C09133=1217.822,182.147,-55.204,-177.681,6.059,148.397
C09134=1217.818,182.396,-55.226,-177.678,6.061,148.396
C09135=1217.814,182.645,-55.250,-177.676,6.062,148.396
C09136=1217.809,182.894,-55.272,-177.674,6.064,148.396
C09137=1217.804,183.143,-55.295,-177.670,6.066,148.395
C09138=1217.799,183.392,-55.318,-177.668,6.067,148.395
C09139=1217.795,183.641,-55.340,-177.666,6.068,148.394
C09140=1217.790,183.890,-55.364,-177.663,6.070,148.394
C09141=1217.785,184.139,-55.387,-177.660,6.072,148.394
C09142=1217.781,184.387,-55.409,-177.658,6.074,148.393
C09143=1217.776,184.636,-55.433,-177.655,6.075,148.393
C09144=1217.772,184.886,-55.455,-177.652,6.076,148.392
C09145=1217.767,185.155,-55.480,-177.650,6.078,148.392
C09146=1217.762,185.425,-55.506,-177.647,6.080,148.392
C09147=1217.757,185.694,-55.530,-177.644,6.082,148.391
C09148=1217.752,185.964,-55.555,-177.641,6.083,148.391
C09149=1217.747,186.213,-55.578,-177.639,6.085,148.390
C09150=1217.742,186.461,-55.600,-177.636,6.087,148.390
C09151=1217.738,186.710,-55.623,-177.634,6.088,148.390
C09152=1217.733,186.960,-55.647,-177.631,6.090,148.389
C09153=1217.728,187.209,-55.670,-177.628,6.091,148.389
C09154=1217.724,187.457,-55.693,-177.626,6.093,148.388
C09155=1217.720,187.706,-55.716,-177.623,6.095,148.388
C09156=1217.715,187.955,-55.740,-177.621,6.096,148.388
C09157=1217.710,188.203,-55.762,-177.618,6.098,148.387
C09158=1217.706,188.452,-55.785,-177.615,6.100,148.387
C09159=1217.701,188.701,-55.809,-177.613,6.102,148.387
C09160=1217.696,188.950,-55.832,-177.611,6.103,148.386
C09161=1217.692,189.199,-55.855,-177.608,6.104,148.386
C09162=1217.688,189.448,-55.878,-177.605,6.106,148.385
C09163=1217.683,189.697,-55.902,-177.602,6.108,148.385
C09164=1217.678,189.946,-55.925,-177.600,6.110,148.385
C09165=1217.673,190.195,-55.948,-177.598,6.111,148.384
C09166=1217.668,190.444,-55.971,-177.595,6.112,148.384
C09167=1217.664,190.692,-55.994,-177.592,6.114,148.384
C09168=1217.660,190.941,-56.017,-177.590,6.116,148.383
C09169=1217.655,191.190,-56.041,-177.587,6.118,148.383
C09170=1217.650,191.439,-56.064,-177.585,6.119,148.382
C09171=1217.645,191.688,-56.088,-177.582,6.120,148.382
C09172=1217.641,191.938,-56.111,-177.579,6.122,148.382
C09173=1217.637,192.186,-56.134,-177.576,6.124,148.381
C09174=1217.632,192.435,-56.158,-177.574,6.126,148.381
C09175=1217.628,192.684,-56.181,-177.572,6.127,148.380
C09176=1217.622,192.932,-56.204,-177.569,6.129,148.380
C09177=1217.618,193.181,-56.227,-177.566,6.131,148.380
C09178=1217.613,193.430,-56.251,-177.564,6.132,148.379
C09179=1217.608,193.679,-56.274,-177.561,6.134,148.379
C09180=1217.604,193.928,-56.298,-177.559,6.135,148.379
C09181=1217.599,194.177,-56.322,-177.556,6.137,148.378
C09182=1217.595,194.425,-56.344,-177.553,6.139,148.378
C09183=1217.591,194.674,-56.368,-177.551,6.140,148.377
C09184=1217.586,194.923,-56.391,-177.548,6.142,148.377
C09185=1217.581,195.172,-56.415,-177.545,6.144,148.377
C09186=1217.577,195.421,-56.439,-177.543,6.145,148.376
C09187=1217.572,195.670,-56.462,-177.541,6.147,148.376
C09188=1217.567,195.919,-56.485,-177.538,6.149,148.376
C09189=1217.563,196.167,-56.509,-177.535,6.151,148.375
C09190=1217.558,196.416,-56.533,-177.533,6.152,148.375
C09191=1217.554,196.665,-56.556,-177.530,6.154,148.375
C09192=1217.549,196.914,-56.580,-177.528,6.155,148.374
C09193=1217.544,197.163,-56.603,-177.525,6.157,148.374
C09194=1217.540,197.412,-56.627,-177.523,6.159,148.374
C09195=1217.535,197.660,-56.651,-177.520,6.161,148.373
C09196=1217.531,197.909,-56.674,-177.517,6.163,148.373
C09197=1217.526,198.158,-56.698,-177.514,6.164,148.372
C09198=1217.522,198.407,-56.722,-177.512,6.165,148.372
C09199=1217.517,198.656,-56.745,-177.510,6.167,148.372
C09200=1217.512,198.905,-56.768,-177.507,6.169,148.371
C09201=1217.508,199.153,-56.792,-177.504,6.171,148.371
C09202=1217.504,199.403,-56.816,-177.502,6.173,148.371
C09203=1217.499,199.651,-56.840,-177.499,6.174,148.370
C09204=1217.494,199.901,-56.864,-177.497,6.175,148.370
C09205=1217.489,200.149,-56.888,-177.494,6.177,148.370
C09206=1217.485,200.398,-56.912,-177.492,6.179,148.369
C09207=1217.480,200.647,-56.936,-177.489,6.181,148.369
C09208=1217.476,200.896,-56.959,-177.486,6.183,148.368
C09209=1217.471,201.144,-56.983,-177.484,6.185,148.368
C09210=1217.467,201.393,-57.007,-177.481,6.186,148.368
C09211=1217.462,201.641,-57.031,-177.478,6.188,148.367
C09212=1217.457,201.890,-57.054,-177.476,6.189,148.367
C09213=1217.452,202.139,-57.079,-177.474,6.191,148.367
C09214=1217.448,202.389,-57.102,-177.471,6.193,148.366
C09215=1217.444,202.637,-57.126,-177.468,6.195,148.366
C09216=1217.439,202.886,-57.150,-177.466,6.197,148.366
C09217=1217.435,203.135,-57.174,-177.463,6.198,148.365
C09218=1217.430,203.383,-57.198,-177.460,6.200,148.365
C09219=1217.425,203.633,-57.222,-177.458,6.202,148.365
C09220=1217.421,203.881,-57.246,-177.456,6.203,148.364
C09221=1217.416,204.130,-57.269,-177.453,6.205,148.364
C09222=1217.412,204.379,-57.294,-177.450,6.207,148.364
C09223=1217.408,204.627,-57.318,-177.448,6.209,148.363
C09224=1217.402,204.877,-57.342,-177.445,6.211,148.363
C09225=1217.398,205.125,-57.366,-177.442,6.212,148.363
C09226=1217.393,205.374,-57.390,-177.440,6.214,148.362
C09227=1217.389,205.623,-57.413,-177.437,6.216,148.362
C09228=1217.384,205.872,-57.438,-177.435,6.217,148.362
C09229=1217.380,206.121,-57.462,-177.432,6.219,148.361
C09230=1217.375,206.370,-57.486,-177.429,6.220,148.361
C09231=1217.371,206.618,-57.510,-177.427,6.222,148.360
C09232=1217.366,206.867,-57.535,-177.424,6.224,148.360
C09233=1217.362,207.116,-57.559,-177.421,6.226,148.360
C09234=1217.357,207.365,-57.582,-177.419,6.228,148.359
C09235=1217.352,207.614,-57.607,-177.417,6.230,148.359
C09236=1217.348,207.862,-57.631,-177.414,6.232,148.359
C09237=1217.343,208.110,-57.655,-177.411,6.234,148.359
C09238=1217.339,208.359,-57.680,-177.409,6.235,148.358
C09239=1217.334,208.609,-57.704,-177.407,6.236,148.358
C09240=1217.330,208.857,-57.728,-177.404,6.238,148.358
C09241=1217.324,209.106,-57.752,-177.401,6.240,148.357
C09242=1217.320,209.354,-57.776,-177.399,6.242,148.357
C09243=1217.316,209.603,-57.801,-177.396,6.244,148.357
C09244=1217.311,209.852,-57.825,-177.393,6.246,148.356
C09245=1217.307,210.101,-57.850,-177.391,6.248,148.356
C09246=1217.302,210.349,-57.874,-177.388,6.249,148.355
C09247=1217.297,210.599,-57.898,-177.386,6.251,148.355
C09248=1217.293,210.848,-57.922,-177.383,6.253,148.355
C09249=1217.288,211.118,-57.949,-177.380,6.255,148.354
C09250=1217.283,211.388,-57.975,-177.377,6.256,148.354
C09251=1217.278,211.659,-58.002,-177.375,6.258,148.354
C09252=1217.273,211.929,-58.028,-177.372,6.260,148.353
C09253=1217.268,212.178,-58.053,-177.369,6.262,148.353
C09254=1217.264,212.426,-58.077,-177.367,6.264,148.353
C09255=1217.259,212.676,-58.102,-177.364,6.266,148.352
C09256=1217.255,212.924,-58.126,-177.361,6.268,148.352
C09257=1217.250,213.173,-58.150,-177.359,6.269,148.352
C09258=1217.246,213.422,-58.175,-177.356,6.271,148.351
C09259=1217.241,213.671,-58.200,-177.353,6.273,148.351
C09260=1217.237,213.919,-58.224,-177.351,6.275,148.351
C09261=1217.232,214.168,-58.249,-177.348,6.277,148.350
C09262=1217.228,214.416,-58.273,-177.346,6.279,148.350
C09263=1217.223,214.665,-58.298,-177.343,6.281,148.350
C09264=1217.219,214.914,-58.323,-177.341,6.283,148.349
C09265=1217.214,215.163,-58.347,-177.338,6.285,148.349
C09266=1217.209,215.411,-58.371,-177.335,6.286,148.349
C09267=1217.205,215.661,-58.396,-177.333,6.288,148.348
C09268=1217.201,215.909,-58.420,-177.330,6.290,148.348
C09269=1217.195,216.158,-58.445,-177.328,6.292,148.348
C09270=1217.192,216.406,-58.470,-177.325,6.294,148.347
C09271=1217.187,216.655,-58.495,-177.322,6.296,148.347
C09272=1217.182,216.904,-58.519,-177.320,6.297,148.347
C09273=1217.178,217.153,-58.544,-177.318,6.298,148.346
C09274=1217.173,217.402,-58.569,-177.315,6.300,148.346
C09275=1217.169,217.650,-58.594,-177.312,6.302,148.346
C09276=1217.164,217.899,-58.618,-177.310,6.304,148.345
C09277=1217.160,218.147,-58.643,-177.307,6.306,148.345
C09278=1217.155,218.397,-58.668,-177.305,6.308,148.345
C09279=1217.150,218.645,-58.693,-177.302,6.310,148.345
C09280=1217.147,218.894,-58.717,-177.300,6.312,148.344
C09281=1217.141,219.143,-58.742,-177.297,6.314,148.344
C09282=1217.136,219.391,-58.767,-177.294,6.315,148.344
C09283=1217.133,219.640,-58.792,-177.292,6.317,148.343
C09284=1217.128,219.889,-58.817,-177.289,6.319,148.343
C09285=1217.123,220.138,-58.842,-177.286,6.321,148.343
C09286=1217.119,220.386,-58.866,-177.284,6.323,148.342
C09287=1217.115,220.635,-58.891,-177.281,6.325,148.342
C09288=1217.109,220.884,-58.916,-177.279,6.327,148.342
C09289=1217.105,221.132,-58.941,-177.276,6.329,148.342
C09290=1217.101,221.381,-58.966,-177.274,6.331,148.341
C09291=1217.096,221.629,-58.991,-177.271,6.332,148.341
C09292=1217.092,221.878,-59.016,-177.269,6.334,148.341
C09293=1217.087,222.127,-59.040,-177.266,6.336,148.340
C09294=1217.083,222.376,-59.066,-177.263,6.338,148.340
C09295=1217.078,222.625,-59.091,-177.261,6.340,148.340
C09296=1217.074,222.873,-59.116,-177.258,6.342,148.339
C09297=1217.069,223.122,-59.141,-177.255,6.344,148.339
C09298=1217.065,223.371,-59.166,-177.253,6.346,148.339
C09299=1217.060,223.619,-59.191,-177.251,6.348,148.339
C09300=1217.056,223.868,-59.216,-177.248,6.349,148.338
C09301=1217.051,224.117,-59.241,-177.245,6.351,148.338
C09302=1217.047,224.365,-59.267,-177.243,6.353,148.338
C09303=1217.042,224.614,-59.291,-177.240,6.355,148.337
C09304=1217.038,224.863,-59.317,-177.237,6.357,148.337
C09305=1217.033,225.111,-59.341,-177.235,6.359,148.337
C09306=1217.029,225.360,-59.367,-177.233,6.361,148.337
C09307=1217.024,225.609,-59.392,-177.230,6.363,148.336
C09308=1217.020,225.858,-59.417,-177.227,6.365,148.336
C09309=1217.014,226.106,-59.442,-177.225,6.366,148.336
C09310=1217.010,226.355,-59.468,-177.222,6.368,148.335
C09311=1217.005,226.603,-59.493,-177.219,6.370,148.335
C09312=1217.002,226.852,-59.518,-177.217,6.372,148.335
C09313=1216.997,227.101,-59.543,-177.215,6.374,148.334
C09314=1216.993,227.349,-59.569,-177.212,6.376,148.334
C09315=1216.988,227.599,-59.594,-177.209,6.378,148.334
C09316=1216.983,227.847,-59.619,-177.207,6.380,148.333
C09317=1216.979,228.096,-59.645,-177.204,6.382,148.333
C09318=1216.974,228.344,-59.670,-177.202,6.383,148.333
C09319=1216.970,228.593,-59.695,-177.199,6.386,148.333
C09320=1216.965,228.842,-59.721,-177.197,6.387,148.332
C09321=1216.961,229.090,-59.745,-177.194,6.389,148.332
C09322=1216.957,229.339,-59.771,-177.192,6.391,148.332
C09323=1216.952,229.587,-59.796,-177.189,6.393,148.331
C09324=1216.948,229.836,-59.822,-177.186,6.395,148.331
C09325=1216.943,230.086,-59.847,-177.184,6.397,148.331
C09326=1216.938,230.334,-59.872,-177.182,6.399,148.331
C09327=1216.934,230.582,-59.898,-177.179,6.401,148.330
C09328=1216.929,230.831,-59.924,-177.176,6.403,148.330
C09329=1216.925,231.079,-59.949,-177.174,6.405,148.330
C09330=1216.921,231.329,-59.974,-177.171,6.406,148.329
C09331=1216.916,231.577,-60.000,-177.169,6.409,148.329
C09332=1216.911,231.826,-60.026,-177.166,6.410,148.329
C09333=1216.907,232.075,-60.051,-177.164,6.412,148.329
C09334=1216.902,232.323,-60.077,-177.161,6.414,148.328
C09335=1216.898,232.571,-60.102,-177.158,6.417,148.328
C09336=1216.894,232.820,-60.128,-177.156,6.419,148.328
C09337=1216.889,233.069,-60.153,-177.153,6.421,148.328
C09338=1216.885,233.318,-60.179,-177.150,6.423,148.327
C09339=1216.880,233.567,-60.205,-177.148,6.425,148.327
C09340=1216.875,233.815,-60.230,-177.145,6.426,148.327
C09341=1216.871,234.064,-60.256,-177.143,6.429,148.327
C09342=1216.866,234.313,-60.282,-177.140,6.430,148.326
C09343=1216.862,234.561,-60.307,-177.138,6.432,148.326
C09344=1216.857,234.809,-60.333,-177.135,6.434,148.326
C09345=1216.853,235.058,-60.359,-177.133,6.436,148.326
C09346=1216.848,235.306,-60.384,-177.130,6.438,148.325
C09347=1216.844,235.555,-60.410,-177.128,6.440,148.325
C09348=1216.840,235.804,-60.436,-177.125,6.442,148.325
C09349=1216.835,236.053,-60.462,-177.122,6.444,148.324
C09350=1216.830,236.301,-60.487,-177.120,6.446,148.324
C09351=1216.826,236.550,-60.513,-177.118,6.448,148.324
C09352=1216.822,236.799,-60.539,-177.115,6.450,148.324
C09353=1216.817,237.069,-60.567,-177.112,6.452,148.323
C09354=1216.812,237.341,-60.595,-177.109,6.454,148.323
C09355=1216.807,237.613,-60.623,-177.107,6.456,148.323
C09356=1216.802,237.884,-60.652,-177.103,6.459,148.322
C09357=1216.797,238.133,-60.678,-177.101,6.461,148.322
C09358=1216.793,238.382,-60.704,-177.099,6.463,148.322
C09359=1216.788,238.630,-60.729,-177.096,6.465,148.322
C09360=1216.784,238.879,-60.755,-177.093,6.467,148.321
C09361=1216.780,239.127,-60.781,-177.091,6.469,148.321
C09362=1216.775,239.376,-60.808,-177.089,6.471,148.321
C09363=1216.771,239.625,-60.833,-177.086,6.473,148.321
C09364=1216.766,239.873,-60.859,-177.083,6.474,148.320
C09365=1216.761,240.122,-60.885,-177.081,6.477,148.320
C09366=1216.757,240.371,-60.911,-177.079,6.478,148.320
C09367=1216.753,240.619,-60.937,-177.076,6.481,148.320
C09368=1216.749,240.868,-60.963,-177.073,6.483,148.319
C09369=1216.743,241.116,-60.989,-177.071,6.485,148.319
C09370=1216.739,241.365,-61.015,-177.068,6.487,148.319
C09371=1216.735,241.613,-61.041,-177.066,6.489,148.319
C09372=1216.730,241.862,-61.068,-177.063,6.491,148.318
C09373=1216.726,242.111,-61.093,-177.061,6.493,148.318
C09374=1216.721,242.359,-61.120,-177.058,6.495,148.318
C09375=1216.716,242.608,-61.146,-177.056,6.497,148.317
C09376=1216.712,242.856,-61.172,-177.053,6.499,148.317
C09377=1216.708,243.105,-61.198,-177.051,6.501,148.317
C09378=1216.703,243.354,-61.224,-177.048,6.503,148.317
C09379=1216.699,243.603,-61.250,-177.045,6.505,148.316
C09380=1216.695,243.851,-61.277,-177.043,6.507,148.316
C09381=1216.690,244.099,-61.303,-177.040,6.509,148.316
C09382=1216.686,244.347,-61.329,-177.038,6.511,148.316
C09383=1216.681,244.596,-61.355,-177.035,6.513,148.316
C09384=1216.676,244.845,-61.381,-177.033,6.515,148.315
C09385=1216.673,245.093,-61.408,-177.030,6.517,148.315
C09386=1216.668,245.343,-61.434,-177.028,6.519,148.315
C09387=1216.664,245.591,-61.460,-177.025,6.521,148.315
C09388=1216.659,245.840,-61.487,-177.022,6.524,148.314
C09389=1216.655,246.088,-61.513,-177.020,6.526,148.314
C09390=1216.650,246.336,-61.539,-177.017,6.528,148.314
C09391=1216.645,246.585,-61.566,-177.015,6.530,148.314
C09392=1216.641,246.833,-61.592,-177.012,6.532,148.313
C09393=1216.636,247.082,-61.619,-177.010,6.534,148.313
C09394=1216.632,247.331,-61.644,-177.007,6.536,148.313
C09395=1216.628,247.579,-61.671,-177.005,6.538,148.313
C09396=1216.623,247.828,-61.697,-177.002,6.541,148.313
C09397=1216.619,248.077,-61.724,-177.000,6.542,148.312
C09398=1216.615,248.325,-61.751,-176.997,6.544,148.312
C09399=1216.610,248.574,-61.777,-176.995,6.547,148.312
C09400=1216.606,248.822,-61.803,-176.992,6.548,148.312
C09401=1216.601,249.071,-61.830,-176.990,6.550,148.311
C09402=1216.597,249.319,-61.856,-176.987,6.552,148.311
C09403=1216.592,249.568,-61.883,-176.985,6.554,148.311
C09404=1216.588,249.817,-61.909,-176.982,6.557,148.311
C09405=1216.583,250.065,-61.936,-176.980,6.559,148.310
C09406=1216.579,250.314,-61.963,-176.977,6.561,148.310
C09407=1216.575,250.562,-61.989,-176.974,6.563,148.310
C09408=1216.570,250.811,-62.016,-176.972,6.565,148.310
C09409=1216.565,251.058,-62.042,-176.970,6.567,148.309
C09410=1216.561,251.307,-62.069,-176.966,6.570,148.309
C09411=1216.557,251.556,-62.095,-176.964,6.572,148.309
C09412=1216.552,251.805,-62.122,-176.962,6.574,148.309
C09413=1216.548,252.053,-62.149,-176.959,6.576,148.308
C09414=1216.544,252.302,-62.176,-176.957,6.578,148.308
C09415=1216.539,252.551,-62.202,-176.954,6.580,148.308
C09416=1216.534,252.799,-62.229,-176.952,6.582,148.308
C09417=1216.530,253.047,-62.256,-176.949,6.585,148.308
C09418=1216.526,253.296,-62.283,-176.946,6.586,148.307
C09419=1216.521,253.544,-62.310,-176.944,6.589,148.307
C09420=1216.517,253.793,-62.336,-176.942,6.591,148.307
C09421=1216.512,254.042,-62.363,-176.939,6.592,148.307
C09422=1216.507,254.290,-62.390,-176.937,6.595,148.307
C09423=1216.504,254.538,-62.416,-176.934,6.597,148.306
C09424=1216.499,254.787,-62.443,-176.931,6.599,148.306
C09425=1216.494,255.035,-62.470,-176.929,6.601,148.306
C09426=1216.490,255.284,-62.497,-176.926,6.603,148.306
C09427=1216.486,255.532,-62.524,-176.924,6.605,148.306
C09428=1216.481,255.781,-62.550,-176.922,6.607,148.305
C09429=1216.476,256.030,-62.577,-176.919,6.610,148.305
C09430=1216.472,256.278,-62.604,-176.916,6.612,148.305
C09431=1216.468,256.527,-62.631,-176.914,6.614,148.305
C09432=1216.463,256.776,-62.658,-176.911,6.616,148.305
C09433=1216.459,257.024,-62.685,-176.909,6.618,148.304
C09434=1216.455,257.272,-62.712,-176.906,6.621,148.304
C09435=1216.450,257.521,-62.739,-176.904,6.623,148.304
C09436=1216.446,257.769,-62.766,-176.901,6.625,148.304
C09437=1216.441,258.018,-62.793,-176.899,6.627,148.303
C09438=1216.436,258.266,-62.820,-176.896,6.629,148.303
C09439=1216.432,258.514,-62.846,-176.893,6.632,148.303
C09440=1216.429,258.763,-62.875,-176.891,6.634,148.303
C09441=1216.424,259.011,-62.902,-176.888,6.636,148.303
C09442=1216.419,259.260,-62.929,-176.886,6.638,148.302
C09443=1216.415,259.508,-62.956,-176.884,6.640,148.302
C09444=1216.410,259.757,-62.983,-176.881,6.643,148.302
C09445=1216.406,260.005,-63.009,-176.878,6.645,148.302
C09446=1216.401,260.254,-63.036,-176.876,6.647,148.302
C09447=1216.397,260.503,-63.064,-176.873,6.649,148.301
C09448=1216.393,260.751,-63.091,-176.871,6.651,148.301
C09449=1216.388,260.999,-63.119,-176.868,6.654,148.301
C09450=1216.384,261.248,-63.146,-176.866,6.656,148.301
C09451=1216.379,261.496,-63.173,-176.863,6.658,148.301
C09452=1216.375,261.745,-63.200,-176.861,6.660,148.300
C09453=1216.370,261.994,-63.227,-176.859,6.662,148.300
C09454=1216.367,262.241,-63.254,-176.856,6.664,148.300
C09455=1216.362,262.490,-63.282,-176.853,6.667,148.300
C09456=1216.357,262.738,-63.309,-176.851,6.669,148.300
C09457=1216.353,263.012,-63.339,-176.848,6.671,148.299
C09458=1216.348,263.284,-63.369,-176.845,6.673,148.299
C09459=1216.343,263.557,-63.399,-176.842,6.676,148.299
C09460=1216.338,263.829,-63.429,-176.840,6.678,148.299
C09461=1216.334,264.077,-63.456,-176.838,6.680,148.299
C09462=1216.330,264.327,-63.483,-176.834,6.683,148.298
C09463=1216.325,264.575,-63.511,-176.832,6.685,148.298
C09464=1216.321,264.823,-63.538,-176.830,6.687,148.298
C09465=1216.316,265.072,-63.565,-176.828,6.689,148.298
C09466=1216.312,265.320,-63.594,-176.824,6.692,148.298
C09467=1216.308,265.569,-63.621,-176.822,6.694,148.298
C09468=1216.303,265.817,-63.648,-176.820,6.696,148.297
C09469=1216.299,266.065,-63.675,-176.817,6.698,148.297
C09470=1216.294,266.315,-63.703,-176.814,6.701,148.297
C09471=1216.289,266.562,-63.731,-176.812,6.703,148.297
C09472=1216.285,266.811,-63.758,-176.810,6.705,148.297
C09473=1216.280,267.059,-63.785,-176.807,6.707,148.297
C09474=1216.276,267.308,-63.814,-176.804,6.710,148.296
C09475=1216.272,267.556,-63.841,-176.802,6.712,148.296
C09476=1216.267,267.804,-63.868,-176.800,6.714,148.296
C09477=1216.263,268.054,-63.896,-176.797,6.716,148.296
C09478=1216.259,268.301,-63.924,-176.794,6.719,148.296
C09479=1216.254,268.550,-63.951,-176.792,6.721,148.296
C09480=1216.251,268.798,-63.979,-176.790,6.723,148.295
C09481=1216.245,269.047,-64.006,-176.787,6.725,148.295
C09482=1216.241,269.295,-64.034,-176.784,6.728,148.295
C09483=1216.236,269.543,-64.062,-176.782,6.730,148.295
C09484=1216.232,269.792,-64.089,-176.779,6.732,148.295
C09485=1216.228,270.040,-64.117,-176.777,6.735,148.294
C09486=1216.224,270.289,-64.145,-176.774,6.737,148.294
C09487=1216.219,270.537,-64.173,-176.772,6.739,148.294
C09488=1216.215,270.785,-64.201,-176.769,6.741,148.294
C09489=1216.210,271.035,-64.228,-176.767,6.744,148.294
C09490=1216.206,271.282,-64.256,-176.764,6.746,148.293
C09491=1216.201,271.531,-64.283,-176.762,6.748,148.293
C09492=1216.197,271.780,-64.312,-176.760,6.750,148.293
C09493=1216.193,272.028,-64.340,-176.757,6.753,148.293
C09494=1216.188,272.276,-64.367,-176.755,6.755,148.293
C09495=1216.184,272.525,-64.395,-176.752,6.757,148.293
C09496=1216.179,272.773,-64.423,-176.749,6.760,148.293
C09497=1216.175,273.022,-64.451,-176.747,6.762,148.292
C09498=1216.171,273.270,-64.478,-176.745,6.764,148.292
C09499=1216.166,273.518,-64.506,-176.742,6.766,148.292
C09500=1216.162,273.767,-64.535,-176.739,6.769,148.292
C09501=1216.158,274.015,-64.563,-176.737,6.771,148.292
C09502=1216.153,274.264,-64.590,-176.735,6.773,148.292
C09503=1216.149,274.512,-64.618,-176.732,6.776,148.292
C09504=1216.145,274.761,-64.647,-176.729,6.778,148.291
C09505=1216.140,275.008,-64.674,-176.727,6.780,148.291
C09506=1216.136,275.256,-64.702,-176.724,6.783,148.291
C09507=1216.131,275.505,-64.731,-176.722,6.785,148.291
C09508=1216.127,275.754,-64.758,-176.720,6.787,148.291
C09509=1216.123,276.002,-64.786,-176.717,6.789,148.291
C09510=1216.118,276.250,-64.814,-176.714,6.792,148.290
C09511=1216.114,276.499,-64.843,-176.712,6.794,148.290
C09512=1216.109,276.747,-64.871,-176.710,6.796,148.290
C09513=1216.105,276.996,-64.899,-176.707,6.799,148.290
C09514=1216.101,277.244,-64.927,-176.704,6.801,148.290
C09515=1216.097,277.493,-64.956,-176.702,6.803,148.290
C09516=1216.092,277.740,-64.983,-176.699,6.806,148.289
C09517=1216.088,277.989,-65.011,-176.697,6.808,148.289
C09518=1216.083,278.237,-65.040,-176.695,6.811,148.289
C09519=1216.080,278.486,-65.068,-176.692,6.813,148.289
C09520=1216.074,278.734,-65.096,-176.690,6.815,148.289
C09521=1216.071,278.983,-65.125,-176.687,6.818,148.289
C09522=1216.066,279.231,-65.153,-176.684,6.820,148.289
C09523=1216.062,279.479,-65.181,-176.682,6.823,148.289
C09524=1216.058,279.727,-65.209,-176.680,6.824,148.288
C09525=1216.053,279.976,-65.238,-176.677,6.827,148.288
C09526=1216.049,280.224,-65.265,-176.675,6.830,148.288
C09527=1216.044,280.473,-65.294,-176.672,6.832,148.288
C09528=1216.040,280.721,-65.322,-176.669,6.835,148.288
C09529=1216.035,280.970,-65.351,-176.667,6.837,148.288
C09530=1216.031,281.218,-65.378,-176.665,6.839,148.288
C09531=1216.027,281.466,-65.407,-176.662,6.842,148.288
C09532=1216.023,281.715,-65.435,-176.660,6.844,148.287
C09533=1216.018,281.963,-65.464,-176.657,6.846,148.287
C09534=1216.014,282.211,-65.492,-176.655,6.849,148.287
C09535=1216.009,282.459,-65.521,-176.653,6.851,148.287
C09536=1216.005,282.708,-65.550,-176.650,6.853,148.287
C09537=1216.000,282.956,-65.577,-176.647,6.856,148.287
C09538=1215.996,283.204,-65.607,-176.645,6.858,148.287
C09539=1215.992,283.453,-65.635,-176.643,6.860,148.286
C09540=1215.987,283.701,-65.663,-176.640,6.863,148.286
C09541=1215.984,283.950,-65.691,-176.638,6.865,148.286
C09542=1215.978,284.198,-65.720,-176.635,6.868,148.286
C09543=1215.974,284.446,-65.749,-176.632,6.870,148.286
C09544=1215.971,284.695,-65.777,-176.630,6.872,148.286
C09545=1215.965,284.943,-65.806,-176.628,6.875,148.286
C09546=1215.961,285.191,-65.835,-176.625,6.877,148.286
C09547=1215.957,285.439,-65.863,-176.623,6.879,148.286
C09548=1215.952,285.688,-65.892,-176.620,6.883,148.286
C09549=1215.948,285.936,-65.921,-176.618,6.884,148.285
C09550=1215.944,286.184,-65.949,-176.616,6.887,148.285
C09551=1215.939,286.433,-65.978,-176.613,6.890,148.285
C09552=1215.935,286.681,-66.007,-176.611,6.892,148.285
C09553=1215.931,286.929,-66.035,-176.608,6.895,148.285
C09554=1215.926,287.178,-66.064,-176.605,6.897,148.285
C09555=1215.922,287.426,-66.093,-176.603,6.899,148.285
C09556=1215.918,287.674,-66.121,-176.600,6.902,148.284
C09557=1215.914,287.922,-66.150,-176.598,6.904,148.284
C09558=1215.909,288.171,-66.179,-176.596,6.906,148.284
C09559=1215.905,288.419,-66.208,-176.593,6.909,148.284
C09560=1215.901,288.667,-66.236,-176.591,6.911,148.284
C09561=1215.896,288.942,-66.268,-176.588,6.914,148.284
C09562=1215.891,289.216,-66.300,-176.585,6.917,148.284
C09563=1215.887,289.490,-66.332,-176.583,6.919,148.284
C09564=1215.882,289.764,-66.364,-176.580,6.922,148.284
C09565=1215.878,290.013,-66.393,-176.577,6.925,148.284
C09566=1215.872,290.261,-66.421,-176.575,6.927,148.283
C09567=1215.868,290.509,-66.451,-176.573,6.929,148.283
C09568=1215.864,290.758,-66.480,-176.570,6.932,148.283
C09569=1215.860,291.006,-66.509,-176.568,6.934,148.283
C09570=1215.855,291.254,-66.537,-176.565,6.937,148.283
C09571=1215.851,291.502,-66.566,-176.563,6.939,148.283
C09572=1215.847,291.751,-66.596,-176.560,6.942,148.283
C09573=1215.842,291.999,-66.625,-176.558,6.945,148.283
C09574=1215.838,292.247,-66.654,-176.556,6.947,148.283
C09575=1215.834,292.495,-66.682,-176.553,6.950,148.283
C09576=1215.830,292.744,-66.711,-176.550,6.952,148.283
C09577=1215.826,292.992,-66.741,-176.548,6.954,148.282
C09578=1215.821,293.240,-66.770,-176.546,6.957,148.282
C09579=1215.816,293.489,-66.798,-176.543,6.959,148.282
C09580=1215.812,293.737,-66.828,-176.541,6.962,148.282
C09581=1215.808,293.985,-66.857,-176.538,6.964,148.282
C09582=1215.803,294.234,-66.886,-176.536,6.966,148.282
C09583=1215.799,294.482,-66.915,-176.533,6.969,148.282
C09584=1215.795,294.729,-66.944,-176.531,6.972,148.282
C09585=1215.791,294.978,-66.974,-176.529,6.975,148.282
C09586=1215.787,295.227,-67.002,-176.526,6.977,148.282
C09587=1215.782,295.475,-67.032,-176.524,6.979,148.282
C09588=1215.778,295.722,-67.061,-176.521,6.982,148.282
C09589=1215.773,295.971,-67.090,-176.519,6.984,148.281
C09590=1215.769,296.219,-67.120,-176.516,6.987,148.281
C09591=1215.765,296.467,-67.149,-176.514,6.989,148.281
C09592=1215.761,296.716,-67.178,-176.512,6.992,148.281
C09593=1215.756,296.964,-67.207,-176.509,6.994,148.281
C09594=1215.752,297.212,-67.236,-176.507,6.996,148.281
C09595=1215.747,297.460,-67.266,-176.504,6.999,148.281
C09596=1215.743,297.709,-67.295,-176.502,7.001,148.281
C09597=1215.739,297.957,-67.325,-176.499,7.005,148.281
C09598=1215.735,298.205,-67.354,-176.497,7.007,148.281
C09599=1215.731,298.453,-67.384,-176.495,7.010,148.281
C09600=1215.726,298.702,-67.413,-176.492,7.012,148.281
C09601=1215.722,298.950,-67.443,-176.490,7.014,148.281
C09602=1215.718,299.197,-67.472,-176.488,7.017,148.281
C09603=1215.713,299.446,-67.501,-176.485,7.019,148.280
C09604=1215.709,299.694,-67.531,-176.482,7.022,148.280
C09605=1215.704,299.943,-67.561,-176.480,7.024,148.280
C09606=1215.700,300.191,-67.590,-176.478,7.027,148.280
C09607=1215.696,300.439,-67.620,-176.476,7.030,148.280
C09608=1215.692,300.687,-67.649,-176.473,7.033,148.280
C09609=1215.688,300.936,-67.678,-176.471,7.035,148.280
C09610=1215.683,301.184,-67.708,-176.469,7.037,148.280
C09611=1215.679,301.432,-67.737,-176.466,7.040,148.280
C09612=1215.675,301.680,-67.767,-176.464,7.042,148.280
C09613=1215.670,301.928,-67.796,-176.461,7.045,148.280
C09614=1215.665,302.177,-67.826,-176.459,7.048,148.280
C09615=1215.661,302.425,-67.855,-176.456,7.051,148.280
C09616=1215.657,302.673,-67.885,-176.454,7.053,148.280
C09617=1215.653,302.921,-67.914,-176.452,7.056,148.280
C09618=1215.649,303.169,-67.945,-176.449,7.058,148.280
C09619=1215.644,303.418,-67.975,-176.447,7.060,148.280
C09620=1215.640,303.666,-68.004,-176.444,7.063,148.280
C09621=1215.636,303.914,-68.033,-176.442,7.065,148.280
C09622=1215.631,304.162,-68.063,-176.439,7.068,148.280
C09623=1215.628,304.410,-68.093,-176.437,7.070,148.280
C09624=1215.623,304.659,-68.123,-176.435,7.073,148.280
C09625=1215.618,304.907,-68.153,-176.432,7.076,148.279
C09626=1215.614,305.155,-68.182,-176.430,7.079,148.279
C09627=1215.610,305.403,-68.212,-176.428,7.081,148.279
C09628=1215.605,305.651,-68.242,-176.425,7.084,148.279
C09629=1215.601,305.900,-68.272,-176.423,7.086,148.279
C09630=1215.597,306.148,-68.301,-176.420,7.089,148.279
C09631=1215.592,306.396,-68.332,-176.418,7.091,148.279
C09632=1215.588,306.644,-68.361,-176.416,7.094,148.279
C09633=1215.584,306.892,-68.391,-176.413,7.097,148.279
C09634=1215.580,307.140,-68.421,-176.412,7.099,148.279
C09635=1215.575,307.389,-68.451,-176.409,7.102,148.279
C09636=1215.571,307.637,-68.481,-176.407,7.104,148.279
C09637=1215.567,307.885,-68.511,-176.404,7.107,148.279
C09638=1215.562,308.133,-68.541,-176.402,7.110,148.279
C09639=1215.558,308.381,-68.571,-176.399,7.113,148.279
C09640=1215.554,308.629,-68.601,-176.397,7.115,148.279
C09641=1215.549,308.878,-68.630,-176.395,7.118,148.279
C09642=1215.545,309.125,-68.661,-176.393,7.120,148.279
C09643=1215.541,309.375,-68.691,-176.390,7.123,148.279
C09644=1215.537,309.622,-68.721,-176.388,7.125,148.279
C09645=1215.533,309.870,-68.751,-176.385,7.128,148.279
C09646=1215.528,310.118,-68.781,-176.383,7.131,148.279
C09647=1215.524,310.367,-68.811,-176.381,7.133,148.279
C09648=1215.520,310.615,-68.842,-176.378,7.136,148.279
C09649=1215.515,310.863,-68.871,-176.377,7.138,148.279
C09650=1215.511,311.111,-68.902,-176.374,7.141,148.279
C09651=1215.507,311.359,-68.931,-176.372,7.144,148.279
C09652=1215.503,311.607,-68.961,-176.369,7.147,148.279
C09653=1215.498,311.855,-68.992,-176.367,7.149,148.279
C09654=1215.495,312.104,-69.022,-176.364,7.152,148.279
C09655=1215.490,312.352,-69.053,-176.362,7.154,148.279
C09656=1215.486,312.600,-69.082,-176.359,7.157,148.279
C09657=1215.481,312.848,-69.113,-176.358,7.160,148.279
C09658=1215.477,313.096,-69.143,-176.355,7.163,148.279
C09659=1215.472,313.344,-69.173,-176.353,7.165,148.279
C09660=1215.469,313.592,-69.203,-176.350,7.168,148.279
C09661=1215.465,313.840,-69.235,-176.348,7.170,148.279
C09662=1215.460,314.089,-69.264,-176.346,7.173,148.279
C09663=1215.456,314.337,-69.295,-176.343,7.176,148.279
C09664=1215.452,314.584,-69.325,-176.341,7.179,148.279
C09665=1215.447,314.861,-69.358,-176.339,7.182,148.279
C09666=1215.442,315.136,-69.393,-176.336,7.184,148.279
C09667=1215.437,315.413,-69.426,-176.334,7.187,148.279
C09668=1215.433,315.688,-69.460,-176.331,7.190,148.279
C09669=1215.428,315.936,-69.491,-176.328,7.193,148.279
C09670=1215.424,316.185,-69.520,-176.326,7.195,148.279
C09671=1215.420,316.433,-69.551,-176.324,7.199,148.279
C09672=1215.415,316.681,-69.582,-176.322,7.201,148.279
C09673=1215.412,316.929,-69.612,-176.319,7.204,148.279
C09674=1215.407,317.177,-69.643,-176.317,7.206,148.279
C09675=1215.403,317.425,-69.672,-176.315,7.209,148.279
C09676=1215.399,317.674,-69.704,-176.313,7.212,148.279
C09677=1215.394,317.922,-69.734,-176.310,7.215,148.279
C09678=1215.390,318.169,-69.765,-176.308,7.217,148.279
C09679=1215.386,318.417,-69.795,-176.306,7.220,148.279
C09680=1215.382,318.666,-69.826,-176.304,7.223,148.279
C09681=1215.378,318.914,-69.857,-176.301,7.226,148.279
C09682=1215.373,319.162,-69.887,-176.299,7.228,148.279
C09683=1215.369,319.410,-69.918,-176.296,7.231,148.279
C09684=1215.365,319.658,-69.949,-176.295,7.233,148.280
C09685=1215.360,319.906,-69.979,-176.292,7.237,148.280
C09686=1215.356,320.154,-70.009,-176.290,7.239,148.279
C09687=1215.352,320.403,-70.041,-176.288,7.242,148.280
C09688=1215.348,320.651,-70.071,-176.286,7.244,148.280
C09689=1215.343,320.899,-70.102,-176.283,7.247,148.280
C09690=1215.339,321.147,-70.132,-176.281,7.250,148.280
C09691=1215.335,321.395,-70.163,-176.279,7.253,148.280
C09692=1215.331,321.643,-70.194,-176.277,7.255,148.280
C09693=1215.326,321.890,-70.225,-176.274,7.258,148.280
C09694=1215.322,322.139,-70.256,-176.272,7.261,148.280
C09695=1215.319,322.387,-70.286,-176.270,7.264,148.280
C09696=1215.314,322.635,-70.317,-176.267,7.266,148.280
C09697=1215.310,322.883,-70.348,-176.265,7.269,148.280
C09698=1215.305,323.131,-70.379,-176.263,7.272,148.280
C09699=1215.301,323.379,-70.410,-176.261,7.275,148.280
C09700=1215.297,323.627,-70.440,-176.259,7.277,148.280
C09701=1215.293,323.875,-70.471,-176.256,7.280,148.280
C09702=1215.289,324.123,-70.503,-176.255,7.283,148.280
C09703=1215.285,324.371,-70.534,-176.252,7.286,148.280
C09704=1215.280,324.619,-70.564,-176.250,7.288,148.280
C09705=1215.275,324.867,-70.595,-176.248,7.291,148.281
C09706=1215.272,325.116,-70.626,-176.245,7.293,148.281
C09707=1215.268,325.363,-70.657,-176.243,7.297,148.281
C09708=1215.263,325.611,-70.688,-176.241,7.299,148.281
C09709=1215.259,325.860,-70.719,-176.238,7.302,148.281
C09710=1215.254,326.108,-70.750,-176.237,7.305,148.281
C09711=1215.250,326.356,-70.781,-176.234,7.308,148.281
C09712=1215.246,326.604,-70.813,-176.233,7.310,148.281
C09713=1215.242,326.852,-70.843,-176.230,7.313,148.281
C09714=1215.238,327.100,-70.874,-176.228,7.316,148.281
C09715=1215.234,327.347,-70.905,-176.226,7.319,148.281
C09716=1215.230,327.596,-70.936,-176.223,7.321,148.281
C09717=1215.225,327.844,-70.967,-176.221,7.324,148.281
C09718=1215.221,328.091,-70.999,-176.219,7.327,148.281
C09719=1215.217,328.340,-71.030,-176.217,7.330,148.282
C09720=1215.212,328.588,-71.061,-176.215,7.332,148.282
C09721=1215.209,328.836,-71.092,-176.213,7.335,148.282
C09722=1215.204,329.084,-71.123,-176.211,7.338,148.282
C09723=1215.200,329.332,-71.155,-176.208,7.341,148.282
C09724=1215.196,329.580,-71.186,-176.206,7.343,148.282
C09725=1215.191,329.828,-71.217,-176.204,7.347,148.282
C09726=1215.187,330.076,-71.248,-176.202,7.349,148.282
C09727=1215.183,330.324,-71.279,-176.200,7.352,148.282
C09728=1215.179,330.572,-71.311,-176.198,7.354,148.282
C09729=1215.174,330.820,-71.342,-176.195,7.358,148.283
C09730=1215.171,331.068,-71.374,-176.193,7.360,148.282
C09731=1215.166,331.316,-71.404,-176.191,7.363,148.283
C09732=1215.162,331.564,-71.436,-176.189,7.365,148.283
C09733=1215.158,331.812,-71.467,-176.187,7.369,148.283
C09734=1215.154,332.060,-71.499,-176.185,7.371,148.283
C09735=1215.150,332.308,-71.530,-176.182,7.374,148.283
C09736=1215.145,332.556,-71.562,-176.181,7.377,148.283
C09737=1215.140,332.804,-71.593,-176.178,7.380,148.283
C09738=1215.137,333.052,-71.625,-176.176,7.382,148.283
C09739=1215.132,333.300,-71.655,-176.174,7.385,148.283
C09740=1215.128,333.548,-71.687,-176.172,7.388,148.284
C09741=1215.124,333.795,-71.719,-176.171,7.391,148.284
C09742=1215.120,334.044,-71.750,-176.168,7.394,148.284
C09743=1215.116,334.291,-71.781,-176.166,7.396,148.284
C09744=1215.112,334.539,-71.813,-176.164,7.399,148.284
C09745=1215.107,334.788,-71.845,-176.162,7.402,148.284
C09746=1215.103,335.036,-71.876,-176.160,7.405,148.284
C09747=1215.099,335.283,-71.908,-176.158,7.407,148.284
C09748=1215.095,335.532,-71.939,-176.155,7.411,148.285
C09749=1215.090,335.779,-71.970,-176.154,7.413,148.285
C09750=1215.087,336.027,-72.002,-176.151,7.416,148.285
C09751=1215.082,336.276,-72.034,-176.149,7.419,148.285
C09752=1215.078,336.523,-72.066,-176.147,7.422,148.285
C09753=1215.074,336.772,-72.097,-176.145,7.424,148.285
C09754=1215.070,337.019,-72.129,-176.143,7.428,148.285
C09755=1215.066,337.268,-72.160,-176.141,7.430,148.285
C09756=1215.061,337.515,-72.192,-176.139,7.433,148.286
C09757=1215.057,337.763,-72.224,-176.137,7.436,148.286
C09758=1215.053,338.011,-72.256,-176.135,7.439,148.286
C09759=1215.049,338.259,-72.287,-176.133,7.442,148.286
C09760=1215.044,338.508,-72.319,-176.130,7.445,148.286
C09761=1215.040,338.755,-72.350,-176.129,7.447,148.286
C09762=1215.036,339.003,-72.382,-176.127,7.450,148.286
C09763=1215.032,339.251,-72.414,-176.125,7.453,148.287
C09764=1215.027,339.499,-72.446,-176.122,7.456,148.287
C09765=1215.024,339.747,-72.478,-176.121,7.459,148.287
C09766=1215.020,339.995,-72.510,-176.118,7.462,148.287
C09767=1215.015,340.242,-72.542,-176.117,7.464,148.287
C09768=1215.011,340.491,-72.573,-176.115,7.468,148.287
C09769=1215.007,340.769,-72.609,-176.112,7.471,148.287
C09770=1215.002,341.046,-72.645,-176.110,7.473,148.288
C09771=1214.997,341.324,-72.681,-176.108,7.477,148.288
C09772=1214.992,341.602,-72.716,-176.106,7.480,148.288
C09773=1214.988,341.850,-72.748,-176.103,7.483,148.288
C09774=1214.984,342.099,-72.780,-176.102,7.486,148.288
C09775=1214.979,342.346,-72.812,-176.099,7.489,148.289
C09776=1214.976,342.594,-72.844,-176.098,7.492,148.289
C09777=1214.971,342.842,-72.876,-176.096,7.495,148.289
C09778=1214.967,343.090,-72.908,-176.094,7.497,148.289
C09779=1214.962,343.338,-72.940,-176.092,7.501,148.289
C09780=1214.959,343.586,-72.972,-176.090,7.503,148.289
C09781=1214.954,343.834,-73.004,-176.088,7.505,148.289
C09782=1214.950,344.081,-73.036,-176.086,7.509,148.290
C09783=1214.947,344.329,-73.068,-176.084,7.511,148.290
C09784=1214.942,344.577,-73.100,-176.082,7.515,148.290
C09785=1214.938,344.825,-73.132,-176.080,7.517,148.290
C09786=1214.933,345.073,-73.165,-176.078,7.521,148.291
C09787=1214.929,345.321,-73.196,-176.076,7.523,148.291
C09788=1214.925,345.569,-73.229,-176.074,7.526,148.291
C09789=1214.921,345.817,-73.260,-176.073,7.529,148.291
C09790=1214.917,346.065,-73.294,-176.070,7.532,148.291
C09791=1214.913,346.312,-73.325,-176.069,7.535,148.291
C09792=1214.908,346.560,-73.357,-176.067,7.538,148.292
C09793=1214.904,346.809,-73.389,-176.065,7.541,148.292
C09794=1214.900,347.057,-73.422,-176.063,7.543,148.292
C09795=1214.896,347.304,-73.454,-176.061,7.546,148.292
C09796=1214.891,347.552,-73.486,-176.059,7.549,148.292
C09797=1214.888,347.800,-73.518,-176.057,7.552,148.293
C09798=1214.883,348.048,-73.551,-176.055,7.555,148.293
C09799=1214.879,348.295,-73.583,-176.053,7.558,148.293
C09800=1214.875,348.543,-73.615,-176.052,7.561,148.293
C09801=1214.871,348.791,-73.647,-176.050,7.564,148.294
C09802=1214.867,349.040,-73.680,-176.048,7.567,148.294
C09803=1214.863,349.286,-73.712,-176.046,7.569,148.294
C09804=1214.858,349.535,-73.744,-176.044,7.573,148.294
C09805=1214.854,349.783,-73.777,-176.042,7.575,148.294
C09806=1214.850,350.031,-73.809,-176.040,7.578,148.295
C09807=1214.846,350.279,-73.842,-176.039,7.581,148.295
C09808=1214.842,350.526,-73.873,-176.036,7.584,148.295
C09809=1214.838,350.774,-73.906,-176.035,7.587,148.295
C09810=1214.833,351.022,-73.939,-176.033,7.589,148.295
C09811=1214.830,351.270,-73.971,-176.031,7.593,148.296
C09812=1214.825,351.518,-74.004,-176.029,7.595,148.296
C09813=1214.820,351.766,-74.036,-176.027,7.599,148.296
C09814=1214.817,352.013,-74.068,-176.026,7.601,148.296
C09815=1214.812,352.262,-74.101,-176.024,7.605,148.297
C09816=1214.808,352.509,-74.134,-176.022,7.607,148.297
C09817=1214.805,352.757,-74.166,-176.020,7.610,148.297
C09818=1214.800,353.005,-74.199,-176.018,7.613,148.297
C09819=1214.795,353.253,-74.231,-176.017,7.616,148.298
C09820=1214.792,353.500,-74.264,-176.015,7.619,148.298
C09821=1214.787,353.748,-74.296,-176.013,7.622,148.298
C09822=1214.783,353.996,-74.329,-176.011,7.625,148.298
C09823=1214.780,354.244,-74.361,-176.009,7.628,148.298
C09824=1214.776,354.492,-74.394,-176.008,7.631,148.299
C09825=1214.771,354.740,-74.427,-176.006,7.634,148.299
C09826=1214.768,354.988,-74.459,-176.004,7.636,148.299
C09827=1214.763,355.235,-74.491,-176.002,7.640,148.299
C09828=1214.758,355.483,-74.524,-176.001,7.643,148.300
C09829=1214.754,355.731,-74.558,-175.999,7.645,148.300
C09830=1214.751,355.979,-74.589,-175.997,7.648,148.300
C09831=1214.747,356.227,-74.623,-175.995,7.651,148.300
C09832=1214.742,356.475,-74.655,-175.994,7.655,148.301
C09833=1214.738,356.723,-74.688,-175.992,7.657,148.301
C09834=1214.734,356.970,-74.721,-175.990,7.660,148.301
C09835=1214.730,357.218,-74.753,-175.989,7.663,148.302
C09836=1214.725,357.465,-74.786,-175.987,7.666,148.302
C09837=1214.721,357.713,-74.819,-175.985,7.668,148.302
C09838=1214.717,357.962,-74.852,-175.984,7.672,148.302
C09839=1214.713,358.209,-74.885,-175.982,7.674,148.303
C09840=1214.709,358.457,-74.917,-175.980,7.678,148.303
C09841=1214.705,358.704,-74.950,-175.979,7.681,148.303
C09842=1214.701,358.953,-74.983,-175.977,7.683,148.303
C09843=1214.696,359.201,-75.016,-175.975,7.687,148.304
C09844=1214.692,359.448,-75.049,-175.974,7.689,148.304
C09845=1214.688,359.696,-75.082,-175.972,7.692,148.304
C09846=1214.685,359.944,-75.114,-175.970,7.696,148.305
C09847=1214.680,360.192,-75.147,-175.968,7.698,148.305
C09848=1214.676,360.439,-75.181,-175.967,7.701,148.305
C09849=1214.672,360.687,-75.214,-175.965,7.704,148.305
C09850=1214.668,360.935,-75.247,-175.963,7.707,148.306
C09851=1214.664,361.183,-75.279,-175.962,7.710,148.306
C09852=1214.659,361.431,-75.312,-175.960,7.713,148.306
C09853=1214.655,361.679,-75.346,-175.959,7.716,148.307
C09854=1214.652,361.926,-75.378,-175.957,7.719,148.307
C09855=1214.648,362.174,-75.411,-175.955,7.722,148.307
C09856=1214.644,362.422,-75.444,-175.954,7.724,148.307
C09857=1214.639,362.669,-75.478,-175.953,7.727,148.308
C09858=1214.635,362.917,-75.511,-175.950,7.731,148.308
C09859=1214.631,363.165,-75.543,-175.949,7.733,148.309
C09860=1214.627,363.413,-75.576,-175.948,7.736,148.309
C09861=1214.623,363.661,-75.610,-175.946,7.740,148.309
C09862=1214.618,363.909,-75.643,-175.945,7.742,148.310
C09863=1214.614,364.156,-75.676,-175.943,7.745,148.310
C09864=1214.610,364.404,-75.709,-175.941,7.749,148.310
C09865=1214.606,364.652,-75.742,-175.940,7.751,148.310
C09866=1214.602,364.900,-75.775,-175.938,7.754,148.311
C09867=1214.598,365.147,-75.808,-175.937,7.757,148.311
C09868=1214.594,365.395,-75.842,-175.935,7.760,148.311
C09869=1214.589,365.643,-75.875,-175.934,7.763,148.312
C09870=1214.585,365.890,-75.908,-175.932,7.765,148.312
C09871=1214.581,366.138,-75.941,-175.931,7.768,148.312
C09872=1214.577,366.386,-75.974,-175.929,7.772,148.313
C09873=1214.573,366.666,-76.012,-175.928,7.775,148.313
C09874=1214.568,366.946,-76.050,-175.926,7.778,148.313
C09875=1214.564,367.226,-76.086,-175.924,7.782,148.314
C09876=1214.559,367.507,-76.125,-175.923,7.784,148.314
C09877=1214.555,367.754,-76.158,-175.921,7.788,148.315
C09878=1214.551,368.002,-76.191,-175.920,7.791,148.315
C09879=1214.546,368.250,-76.224,-175.918,7.793,148.315
C09880=1214.542,368.498,-76.258,-175.917,7.796,148.316
C09881=1214.538,368.745,-76.291,-175.916,7.799,148.316
C09882=1214.534,368.992,-76.325,-175.914,7.802,148.316
C09883=1214.530,369.240,-76.358,-175.913,7.805,148.317
C09884=1214.526,369.488,-76.391,-175.911,7.808,148.317
C09885=1214.522,369.736,-76.424,-175.910,7.811,148.317
C09886=1214.518,369.984,-76.458,-175.909,7.814,148.318
C09887=1214.514,370.231,-76.492,-175.907,7.817,148.318
C09888=1214.510,370.479,-76.525,-175.906,7.820,148.319
C09889=1214.505,370.727,-76.558,-175.904,7.823,148.319
C09890=1214.501,370.975,-76.592,-175.903,7.826,148.319
C09891=1214.497,371.222,-76.625,-175.902,7.828,148.320
C09892=1214.493,371.469,-76.659,-175.901,7.831,148.320
C09893=1214.489,371.717,-76.692,-175.900,7.834,148.320
C09894=1214.485,371.966,-76.726,-175.898,7.838,148.321
C09895=1214.481,372.214,-76.759,-175.896,7.840,148.321
C09896=1214.477,372.461,-76.793,-175.895,7.843,148.322
C09897=1214.473,372.708,-76.826,-175.894,7.846,148.322
C09898=1214.469,372.956,-76.859,-175.893,7.849,148.322
C09899=1214.464,373.204,-76.894,-175.892,7.851,148.323
C09900=1214.460,373.451,-76.927,-175.890,7.854,148.323
C09901=1214.456,373.700,-76.960,-175.889,7.857,148.323
C09902=1214.453,373.947,-76.994,-175.888,7.860,148.324
C09903=1214.449,374.195,-77.027,-175.887,7.863,148.324
C09904=1214.444,374.443,-77.061,-175.886,7.865,148.325
C09905=1214.440,374.690,-77.095,-175.884,7.869,148.325
C09906=1214.436,374.937,-77.128,-175.883,7.872,148.325
C09907=1214.432,375.186,-77.162,-175.881,7.875,148.326
C09908=1214.428,375.433,-77.196,-175.880,7.878,148.326
C09909=1214.423,375.681,-77.229,-175.879,7.880,148.327
C09910=1214.420,375.928,-77.263,-175.878,7.883,148.327
C09911=1214.415,376.176,-77.296,-175.877,7.886,148.327
C09912=1214.411,376.425,-77.330,-175.875,7.889,148.328
C09913=1214.407,376.672,-77.364,-175.874,7.892,148.328
C09914=1214.403,376.919,-77.397,-175.873,7.894,148.329
C09915=1214.399,377.167,-77.431,-175.872,7.897,148.329
C09916=1214.394,377.415,-77.465,-175.871,7.900,148.329
C09917=1214.391,377.662,-77.499,-175.870,7.903,148.330
C09918=1214.387,377.910,-77.532,-175.869,7.906,148.330
C09919=1214.383,378.158,-77.567,-175.868,7.909,148.331
C09920=1214.378,378.405,-77.600,-175.866,7.912,148.331
C09921=1214.375,378.652,-77.634,-175.865,7.914,148.332
C09922=1214.370,378.901,-77.668,-175.864,7.917,148.332
C09923=1214.366,379.148,-77.702,-175.863,7.919,148.332
C09924=1214.362,379.396,-77.735,-175.863,7.922,148.333
C09925=1214.358,379.643,-77.770,-175.861,7.925,148.333
C09926=1214.354,379.892,-77.803,-175.860,7.928,148.334
C09927=1214.350,380.139,-77.837,-175.859,7.931,148.334
C09928=1214.346,380.387,-77.871,-175.858,7.934,148.334
C09929=1214.342,380.634,-77.905,-175.857,7.936,148.335
C09930=1214.338,380.883,-77.938,-175.856,7.940,148.335
C09931=1214.334,381.130,-77.973,-175.855,7.942,148.336
C09932=1214.330,381.377,-78.006,-175.854,7.945,148.336
C09933=1214.325,381.625,-78.040,-175.852,7.948,148.337
C09934=1214.322,381.873,-78.074,-175.852,7.950,148.337
C09935=1214.318,382.121,-78.108,-175.851,7.953,148.338
C09936=1214.313,382.368,-78.142,-175.850,7.956,148.338
C09937=1214.309,382.615,-78.176,-175.849,7.959,148.338
C09938=1214.305,382.864,-78.210,-175.848,7.962,148.339
C09939=1214.301,383.111,-78.244,-175.847,7.965,148.339
C09940=1214.297,383.358,-78.278,-175.846,7.967,148.340
C09941=1214.292,383.606,-78.312,-175.845,7.970,148.340
C09942=1214.289,383.854,-78.346,-175.844,7.973,148.341
C09943=1214.284,384.101,-78.380,-175.843,7.975,148.341
C09944=1214.280,384.349,-78.413,-175.842,7.978,148.341
C09945=1214.276,384.597,-78.448,-175.841,7.980,148.342
C09946=1214.273,384.844,-78.482,-175.840,7.983,148.342
C09947=1214.268,385.092,-78.515,-175.839,7.986,148.343
C09948=1214.264,385.340,-78.550,-175.838,7.989,148.343
C09949=1214.261,385.587,-78.584,-175.837,7.992,148.344
C09950=1214.256,385.835,-78.618,-175.836,7.994,148.344
C09951=1214.252,386.082,-78.652,-175.836,7.997,148.345
C09952=1214.248,386.331,-78.686,-175.835,8.000,148.345
C09953=1214.244,386.578,-78.720,-175.834,8.003,148.346
C09954=1214.240,386.825,-78.755,-175.833,8.005,148.346
C09955=1214.236,387.074,-78.788,-175.832,8.008,148.346
C09956=1214.231,387.321,-78.823,-175.831,8.011,148.347
C09957=1214.228,387.568,-78.857,-175.831,8.013,148.347
C09958=1214.224,387.816,-78.891,-175.829,8.016,148.348
C09959=1214.220,388.063,-78.925,-175.829,8.019,148.348
C09960=1214.215,388.311,-78.959,-175.828,8.021,148.349
C09961=1214.212,388.559,-78.993,-175.827,8.024,148.349
C09962=1214.207,388.807,-79.028,-175.826,8.027,148.350
C09963=1214.203,389.054,-79.062,-175.826,8.029,148.350
C09964=1214.199,389.302,-79.096,-175.825,8.032,148.351
C09965=1214.195,389.549,-79.130,-175.823,8.035,148.351
C09966=1214.191,389.798,-79.164,-175.823,8.037,148.352
C09967=1214.187,390.045,-79.198,-175.822,8.040,148.352
C09968=1214.183,390.292,-79.233,-175.821,8.043,148.353
C09969=1214.179,390.540,-79.268,-175.821,8.045,148.353
C09970=1214.175,390.787,-79.302,-175.820,8.048,148.354
C09971=1214.170,391.035,-79.336,-175.819,8.050,148.354
C09972=1214.167,391.283,-79.370,-175.819,8.053,148.354
C09973=1214.163,391.530,-79.405,-175.817,8.056,148.355
C09974=1214.159,391.778,-79.438,-175.817,8.058,148.355
C09975=1214.155,392.026,-79.473,-175.816,8.061,148.356
C09976=1214.150,392.273,-79.507,-175.815,8.063,148.356
C09977=1214.146,392.555,-79.546,-175.815,8.066,148.357
C09978=1214.141,392.838,-79.585,-175.814,8.069,148.357
C09979=1214.136,393.119,-79.625,-175.813,8.072,148.358
C09980=1214.132,393.402,-79.664,-175.812,8.075,148.358
C09981=1214.128,393.649,-79.698,-175.812,8.077,148.359
C09982=1214.124,393.897,-79.732,-175.810,8.080,148.359
C09983=1214.120,394.145,-79.766,-175.810,8.082,148.360
C09984=1214.116,394.392,-79.801,-175.809,8.085,148.360
C09985=1214.112,394.640,-79.836,-175.809,8.087,148.361
C09986=1214.108,394.887,-79.869,-175.808,8.090,148.361
C09987=1214.104,395.135,-79.904,-175.807,8.092,148.362
C09988=1214.100,395.382,-79.938,-175.806,8.095,148.362
C09989=1214.095,395.630,-79.973,-175.806,8.098,148.363
C09990=1214.091,395.878,-80.007,-175.805,8.101,148.363
C09991=1214.088,396.124,-80.042,-175.805,8.103,148.364
C09992=1214.084,396.373,-80.077,-175.804,8.106,148.364
C09993=1214.079,396.620,-80.111,-175.803,8.108,148.364
C09994=1214.076,396.867,-80.145,-175.802,8.111,148.365
C09995=1214.072,397.115,-80.180,-175.802,8.113,148.365
C09996=1214.067,397.363,-80.214,-175.802,8.115,148.366
//INST
///DATE 2021/06/25 14:27
///ATTR SC,RW,RJ
////FRAME ROBOT
///GROUP1 RB1
NOP
MOVL C00000 V=800.0 PL=0
MOVL C00001 V=800.0 PL=0
MOVL C00002 V=800.0 PL=0
MOVL C00003 V=800.0 PL=0
MOVL C00004 V=800.0 PL=0
MOVL C00005 V=800.0 PL=0
MOVL C00006 V=800.0 PL=0
MOVL C00007 V=800.0 PL=0
MOVL C00008 V=800.0 PL=0
MOVL C00009 V=800.0 PL=0
MOVL C00010 V=800.0 PL=0
MOVL C00011 V=800.0 PL=0
MOVL C00012 V=800.0 PL=0
MOVL C00013 V=800.0 PL=0
MOVL C00014 V=800.0 PL=0
MOVL C00015 V=800.0 PL=0
MOVL C00016 V=800.0 PL=0
MOVL C00017 V=800.0 PL=0
MOVL C00018 V=800.0 PL=0
MOVL C00019 V=800.0 PL=0
MOVL C00020 V=800.0 PL=0
MOVL C00021 V=800.0 PL=0
MOVL C00022 V=800.0 PL=0
MOVL C00023 V=800.0 PL=0
MOVL C00024 V=800.0 PL=0
MOVL C00025 V=800.0 PL=0
MOVL C00026 V=800.0 PL=0
MOVL C00027 V=800.0 PL=0
MOVL C00028 V=800.0 PL=0
MOVL C00029 V=800.0 PL=0
MOVL C00030 V=800.0 PL=0
MOVL C00031 V=800.0 PL=0
MOVL C00032 V=800.0 PL=0
MOVL C00033 V=800.0 PL=0
MOVL C00034 V=800.0 PL=0
MOVL C00035 V=800.0 PL=0
MOVL C00036 V=800.0 PL=0
MOVL C00037 V=800.0 PL=0
MOVL C00038 V=800.0 PL=0
MOVL C00039 V=800.0 PL=0
MOVL C00040 V=800.0 PL=0
MOVL C00041 V=800.0 PL=0
MOVL C00042 V=800.0 PL=0
MOVL C00043 V=800.0 PL=0
MOVL C00044 V=800.0 PL=0
MOVL C00045 V=800.0 PL=0
MOVL C00046 V=800.0 PL=0
MOVL C00047 V=800.0 PL=0
MOVL C00048 V=800.0 PL=0
MOVL C00049 V=800.0 PL=0
MOVL C00050 V=800.0 PL=0
MOVL C00051 V=800.0 PL=0
MOVL C00052 V=800.0 PL=0
MOVL C00053 V=800.0 PL=0
MOVL C00054 V=800.0 PL=0
MOVL C00055 V=800.0 PL=0
MOVL C00056 V=800.0 PL=0
MOVL C00057 V=800.0 PL=0
MOVL C00058 V=800.0 PL=0
MOVL C00059 V=800.0 PL=0
MOVL C00060 V=800.0 PL=0
MOVL C00061 V=800.0 PL=0
MOVL C00062 V=800.0 PL=0
MOVL C00063 V=800.0 PL=0
MOVL C00064 V=800.0 PL=0
MOVL C00065 V=800.0 PL=0
MOVL C00066 V=800.0 PL=0
MOVL C00067 V=800.0 PL=0
MOVL C00068 V=800.0 PL=0
MOVL C00069 V=800.0 PL=0
MOVL C00070 V=800.0 PL=0
MOVL C00071 V=800.0 PL=0
MOVL C00072 V=800.0 PL=0
MOVL C00073 V=800.0 PL=0
MOVL C00074 V=800.0 PL=0
MOVL C00075 V=800.0 PL=0
MOVL C00076 V=800.0 PL=0
MOVL C00077 V=800.0 PL=0
MOVL C00078 V=800.0 PL=0
MOVL C00079 V=800.0 PL=0
MOVL C00080 V=800.0 PL=0
MOVL C00081 V=800.0 PL=0
MOVL C00082 V=800.0 PL=0
MOVL C00083 V=800.0 PL=0
MOVL C00084 V=800.0 PL=0
MOVL C00085 V=800.0 PL=0
MOVL C00086 V=800.0 PL=0
MOVL C00087 V=800.0 PL=0
MOVL C00088 V=800.0 PL=0
MOVL C00089 V=800.0 PL=0
MOVL C00090 V=800.0 PL=0
MOVL C00091 V=800.0 PL=0
MOVL C00092 V=800.0 PL=0
MOVL C00093 V=800.0 PL=0
MOVL C00094 V=800.0 PL=0
MOVL C00095 V=800.0 PL=0
MOVL C00096 V=800.0 PL=0
MOVL C00097 V=800.0 PL=0
MOVL C00098 V=800.0 PL=0
MOVL C00099 V=800.0 PL=0
MOVL C00100 V=800.0 PL=0
MOVL C00101 V=800.0 PL=0
MOVL C00102 V=800.0 PL=0
MOVL C00103 V=800.0 PL=0
MOVL C00104 V=800.0 PL=0
MOVL C00105 V=800.0 PL=0
MOVL C00106 V=800.0 PL=0
MOVL C00107 V=800.0 PL=0
MOVL C00108 V=800.0 PL=0
MOVL C00109 V=800.0 PL=0
MOVL C00110 V=800.0 PL=0
MOVL C00111 V=800.0 PL=0
MOVL C00112 V=800.0 PL=0
MOVL C00113 V=800.0 PL=0
MOVL C00114 V=800.0 PL=0
MOVL C00115 V=800.0 PL=0
MOVL C00116 V=800.0 PL=0
MOVL C00117 V=800.0 PL=0
MOVL C00118 V=800.0 PL=0
MOVL C00119 V=800.0 PL=0
MOVL C00120 V=800.0 PL=0
MOVL C00121 V=800.0 PL=0
MOVL C00122 V=800.0 PL=0
MOVL C00123 V=800.0 PL=0
MOVL C00124 V=800.0 PL=0
MOVL C00125 V=800.0 PL=0
MOVL C00126 V=800.0 PL=0
MOVL C00127 V=800.0 PL=0
MOVL C00128 V=800.0 PL=0
MOVL C00129 V=800.0 PL=0
MOVL C00130 V=800.0 PL=0
MOVL C00131 V=800.0 PL=0
MOVL C00132 V=800.0 PL=0
MOVL C00133 V=800.0 PL=0
MOVL C00134 V=800.0 PL=0
MOVL C00135 V=800.0 PL=0
MOVL C00136 V=800.0 PL=0
MOVL C00137 V=800.0 PL=0
MOVL C00138 V=800.0 PL=0
MOVL C00139 V=800.0 PL=0
MOVL C00140 V=800.0 PL=0
MOVL C00141 V=800.0 PL=0
MOVL C00142 V=800.0 PL=0
MOVL C00143 V=800.0 PL=0
MOVL C00144 V=800.0 PL=0
MOVL C00145 V=800.0 PL=0
MOVL C00146 V=800.0 PL=0
MOVL C00147 V=800.0 PL=0
MOVL C00148 V=800.0 PL=0
MOVL C00149 V=800.0 PL=0
MOVL C00150 V=800.0 PL=0
MOVL C00151 V=800.0 PL=0
MOVL C00152 V=800.0 PL=0
MOVL C00153 V=800.0 PL=0
MOVL C00154 V=800.0 PL=0
MOVL C00155 V=800.0 PL=0
MOVL C00156 V=800.0 PL=0
MOVL C00157 V=800.0 PL=0
MOVL C00158 V=800.0 PL=0
MOVL C00159 V=800.0 PL=0
MOVL C00160 V=800.0 PL=0
MOVL C00161 V=800.0 PL=0
MOVL C00162 V=800.0 PL=0
MOVL C00163 V=800.0 PL=0
MOVL C00164 V=800.0 PL=0
MOVL C00165 V=800.0 PL=0
MOVL C00166 V=800.0 PL=0
MOVL C00167 V=800.0 PL=0
MOVL C00168 V=800.0 PL=0
MOVL C00169 V=800.0 PL=0
MOVL C00170 V=800.0 PL=0
MOVL C00171 V=800.0 PL=0
MOVL C00172 V=800.0 PL=0
MOVL C00173 V=800.0 PL=0
MOVL C00174 V=800.0 PL=0
MOVL C00175 V=800.0 PL=0
MOVL C00176 V=800.0 PL=0
MOVL C00177 V=800.0 PL=0
MOVL C00178 V=800.0 PL=0
MOVL C00179 V=800.0 PL=0
MOVL C00180 V=800.0 PL=0
MOVL C00181 V=800.0 PL=0
MOVL C00182 V=800.0 PL=0
MOVL C00183 V=800.0 PL=0
MOVL C00184 V=800.0 PL=0
MOVL C00185 V=800.0 PL=0
MOVL C00186 V=800.0 PL=0
MOVL C00187 V=800.0 PL=0
MOVL C00188 V=800.0 PL=0
MOVL C00189 V=800.0 PL=0
MOVL C00190 V=800.0 PL=0
MOVL C00191 V=800.0 PL=0
MOVL C00192 V=800.0 PL=0
MOVL C00193 V=800.0 PL=0
MOVL C00194 V=800.0 PL=0
MOVL C00195 V=800.0 PL=0
MOVL C00196 V=800.0 PL=0
MOVL C00197 V=800.0 PL=0
MOVL C00198 V=800.0 PL=0
MOVL C00199 V=800.0 PL=0
MOVL C00200 V=800.0 PL=0
MOVL C00201 V=800.0 PL=0
MOVL C00202 V=800.0 PL=0
MOVL C00203 V=800.0 PL=0
MOVL C00204 V=800.0 PL=0
MOVL C00205 V=800.0 PL=0
MOVL C00206 V=800.0 PL=0
MOVL C00207 V=800.0 PL=0
MOVL C00208 V=800.0 PL=0
MOVL C00209 V=800.0 PL=0
MOVL C00210 V=800.0 PL=0
MOVL C00211 V=800.0 PL=0
MOVL C00212 V=800.0 PL=0
MOVL C00213 V=800.0 PL=0
MOVL C00214 V=800.0 PL=0
MOVL C00215 V=800.0 PL=0
MOVL C00216 V=800.0 PL=0
MOVL C00217 V=800.0 PL=0
MOVL C00218 V=800.0 PL=0
MOVL C00219 V=800.0 PL=0
MOVL C00220 V=800.0 PL=0
MOVL C00221 V=800.0 PL=0
MOVL C00222 V=800.0 PL=0
MOVL C00223 V=800.0 PL=0
MOVL C00224 V=800.0 PL=0
MOVL C00225 V=800.0 PL=0
MOVL C00226 V=800.0 PL=0
MOVL C00227 V=800.0 PL=0
MOVL C00228 V=800.0 PL=0
MOVL C00229 V=800.0 PL=0
MOVL C00230 V=800.0 PL=0
MOVL C00231 V=800.0 PL=0
MOVL C00232 V=800.0 PL=0
MOVL C00233 V=800.0 PL=0
MOVL C00234 V=800.0 PL=0
MOVL C00235 V=800.0 PL=0
MOVL C00236 V=800.0 PL=0
MOVL C00237 V=800.0 PL=0
MOVL C00238 V=800.0 PL=0
MOVL C00239 V=800.0 PL=0
MOVL C00240 V=800.0 PL=0
MOVL C00241 V=800.0 PL=0
MOVL C00242 V=800.0 PL=0
MOVL C00243 V=800.0 PL=0
MOVL C00244 V=800.0 PL=0
MOVL C00245 V=800.0 PL=0
MOVL C00246 V=800.0 PL=0
MOVL C00247 V=800.0 PL=0
MOVL C00248 V=800.0 PL=0
MOVL C00249 V=800.0 PL=0
MOVL C00250 V=800.0 PL=0
MOVL C00251 V=800.0 PL=0
MOVL C00252 V=800.0 PL=0
MOVL C00253 V=800.0 PL=0
MOVL C00254 V=800.0 PL=0
MOVL C00255 V=800.0 PL=0
MOVL C00256 V=800.0 PL=0
MOVL C00257 V=800.0 PL=0
MOVL C00258 V=800.0 PL=0
MOVL C00259 V=800.0 PL=0
MOVL C00260 V=800.0 PL=0
MOVL C00261 V=800.0 PL=0
MOVL C00262 V=800.0 PL=0
MOVL C00263 V=800.0 PL=0
MOVL C00264 V=800.0 PL=0
MOVL C00265 V=800.0 PL=0
MOVL C00266 V=800.0 PL=0
MOVL C00267 V=800.0 PL=0
MOVL C00268 V=800.0 PL=0
MOVL C00269 V=800.0 PL=0
MOVL C00270 V=800.0 PL=0
MOVL C00271 V=800.0 PL=0
MOVL C00272 V=800.0 PL=0
MOVL C00273 V=800.0 PL=0
MOVL C00274 V=800.0 PL=0
MOVL C00275 V=800.0 PL=0
MOVL C00276 V=800.0 PL=0
MOVL C00277 V=800.0 PL=0
MOVL C00278 V=800.0 PL=0
MOVL C00279 V=800.0 PL=0
MOVL C00280 V=800.0 PL=0
MOVL C00281 V=800.0 PL=0
MOVL C00282 V=800.0 PL=0
MOVL C00283 V=800.0 PL=0
MOVL C00284 V=800.0 PL=0
MOVL C00285 V=800.0 PL=0
MOVL C00286 V=800.0 PL=0
MOVL C00287 V=800.0 PL=0
MOVL C00288 V=800.0 PL=0
MOVL C00289 V=800.0 PL=0
MOVL C00290 V=800.0 PL=0
MOVL C00291 V=800.0 PL=0
MOVL C00292 V=800.0 PL=0
MOVL C00293 V=800.0 PL=0
MOVL C00294 V=800.0 PL=0
MOVL C00295 V=800.0 PL=0
MOVL C00296 V=800.0 PL=0
MOVL C00297 V=800.0 PL=0
MOVL C00298 V=800.0 PL=0
MOVL C00299 V=800.0 PL=0
MOVL C00300 V=800.0 PL=0
MOVL C00301 V=800.0 PL=0
MOVL C00302 V=800.0 PL=0
MOVL C00303 V=800.0 PL=0
MOVL C00304 V=800.0 PL=0
MOVL C00305 V=800.0 PL=0
MOVL C00306 V=800.0 PL=0
MOVL C00307 V=800.0 PL=0
MOVL C00308 V=800.0 PL=0
MOVL C00309 V=800.0 PL=0
MOVL C00310 V=800.0 PL=0
MOVL C00311 V=800.0 PL=0
MOVL C00312 V=800.0 PL=0
MOVL C00313 V=800.0 PL=0
MOVL C00314 V=800.0 PL=0
MOVL C00315 V=800.0 PL=0
MOVL C00316 V=800.0 PL=0
MOVL C00317 V=800.0 PL=0
MOVL C00318 V=800.0 PL=0
MOVL C00319 V=800.0 PL=0
MOVL C00320 V=800.0 PL=0
MOVL C00321 V=800.0 PL=0
MOVL C00322 V=800.0 PL=0
MOVL C00323 V=800.0 PL=0
MOVL C00324 V=800.0 PL=0
MOVL C00325 V=800.0 PL=0
MOVL C00326 V=800.0 PL=0
MOVL C00327 V=800.0 PL=0
MOVL C00328 V=800.0 PL=0
MOVL C00329 V=800.0 PL=0
MOVL C00330 V=800.0 PL=0
MOVL C00331 V=800.0 PL=0
MOVL C00332 V=800.0 PL=0
MOVL C00333 V=800.0 PL=0
MOVL C00334 V=800.0 PL=0
MOVL C00335 V=800.0 PL=0
MOVL C00336 V=800.0 PL=0
MOVL C00337 V=800.0 PL=0
MOVL C00338 V=800.0 PL=0
MOVL C00339 V=800.0 PL=0
MOVL C00340 V=800.0 PL=0
MOVL C00341 V=800.0 PL=0
MOVL C00342 V=800.0 PL=0
MOVL C00343 V=800.0 PL=0
MOVL C00344 V=800.0 PL=0
MOVL C00345 V=800.0 PL=0
MOVL C00346 V=800.0 PL=0
MOVL C00347 V=800.0 PL=0
MOVL C00348 V=800.0 PL=0
MOVL C00349 V=800.0 PL=0
MOVL C00350 V=800.0 PL=0
MOVL C00351 V=800.0 PL=0
MOVL C00352 V=800.0 PL=0
MOVL C00353 V=800.0 PL=0
MOVL C00354 V=800.0 PL=0
MOVL C00355 V=800.0 PL=0
MOVL C00356 V=800.0 PL=0
MOVL C00357 V=800.0 PL=0
MOVL C00358 V=800.0 PL=0
MOVL C00359 V=800.0 PL=0
MOVL C00360 V=800.0 PL=0
MOVL C00361 V=800.0 PL=0
MOVL C00362 V=800.0 PL=0
MOVL C00363 V=800.0 PL=0
MOVL C00364 V=800.0 PL=0
MOVL C00365 V=800.0 PL=0
MOVL C00366 V=800.0 PL=0
MOVL C00367 V=800.0 PL=0
MOVL C00368 V=800.0 PL=0
MOVL C00369 V=800.0 PL=0
MOVL C00370 V=800.0 PL=0
MOVL C00371 V=800.0 PL=0
MOVL C00372 V=800.0 PL=0
MOVL C00373 V=800.0 PL=0
MOVL C00374 V=800.0 PL=0
MOVL C00375 V=800.0 PL=0
MOVL C00376 V=800.0 PL=0
MOVL C00377 V=800.0 PL=0
MOVL C00378 V=800.0 PL=0
MOVL C00379 V=800.0 PL=0
MOVL C00380 V=800.0 PL=0
MOVL C00381 V=800.0 PL=0
MOVL C00382 V=800.0 PL=0
MOVL C00383 V=800.0 PL=0
MOVL C00384 V=800.0 PL=0
MOVL C00385 V=800.0 PL=0
MOVL C00386 V=800.0 PL=0
MOVL C00387 V=800.0 PL=0
MOVL C00388 V=800.0 PL=0
MOVL C00389 V=800.0 PL=0
MOVL C00390 V=800.0 PL=0
MOVL C00391 V=800.0 PL=0
MOVL C00392 V=800.0 PL=0
MOVL C00393 V=800.0 PL=0
MOVL C00394 V=800.0 PL=0
MOVL C00395 V=800.0 PL=0
MOVL C00396 V=800.0 PL=0
MOVL C00397 V=800.0 PL=0
MOVL C00398 V=800.0 PL=0
MOVL C00399 V=800.0 PL=0
MOVL C00400 V=800.0 PL=0
MOVL C00401 V=800.0 PL=0
MOVL C00402 V=800.0 PL=0
MOVL C00403 V=800.0 PL=0
MOVL C00404 V=800.0 PL=0
MOVL C00405 V=800.0 PL=0
MOVL C00406 V=800.0 PL=0
MOVL C00407 V=800.0 PL=0
MOVL C00408 V=800.0 PL=0
MOVL C00409 V=800.0 PL=0
MOVL C00410 V=800.0 PL=0
MOVL C00411 V=800.0 PL=0
MOVL C00412 V=800.0 PL=0
MOVL C00413 V=800.0 PL=0
MOVL C00414 V=800.0 PL=0
MOVL C00415 V=800.0 PL=0
MOVL C00416 V=800.0 PL=0
MOVL C00417 V=800.0 PL=0
MOVL C00418 V=800.0 PL=0
MOVL C00419 V=800.0 PL=0
MOVL C00420 V=800.0 PL=0
MOVL C00421 V=800.0 PL=0
MOVL C00422 V=800.0 PL=0
MOVL C00423 V=800.0 PL=0
MOVL C00424 V=800.0 PL=0
MOVL C00425 V=800.0 PL=0
MOVL C00426 V=800.0 PL=0
MOVL C00427 V=800.0 PL=0
MOVL C00428 V=800.0 PL=0
MOVL C00429 V=800.0 PL=0
MOVL C00430 V=800.0 PL=0
MOVL C00431 V=800.0 PL=0
MOVL C00432 V=800.0 PL=0
MOVL C00433 V=800.0 PL=0
MOVL C00434 V=800.0 PL=0
MOVL C00435 V=800.0 PL=0
MOVL C00436 V=800.0 PL=0
MOVL C00437 V=800.0 PL=0
MOVL C00438 V=800.0 PL=0
MOVL C00439 V=800.0 PL=0
MOVL C00440 V=800.0 PL=0
MOVL C00441 V=800.0 PL=0
MOVL C00442 V=800.0 PL=0
MOVL C00443 V=800.0 PL=0
MOVL C00444 V=800.0 PL=0
MOVL C00445 V=800.0 PL=0
MOVL C00446 V=800.0 PL=0
MOVL C00447 V=800.0 PL=0
MOVL C00448 V=800.0 PL=0
MOVL C00449 V=800.0 PL=0
MOVL C00450 V=800.0 PL=0
MOVL C00451 V=800.0 PL=0
MOVL C00452 V=800.0 PL=0
MOVL C00453 V=800.0 PL=0
MOVL C00454 V=800.0 PL=0
MOVL C00455 V=800.0 PL=0
MOVL C00456 V=800.0 PL=0
MOVL C00457 V=800.0 PL=0
MOVL C00458 V=800.0 PL=0
MOVL C00459 V=800.0 PL=0
MOVL C00460 V=800.0 PL=0
MOVL C00461 V=800.0 PL=0
MOVL C00462 V=800.0 PL=0
MOVL C00463 V=800.0 PL=0
MOVL C00464 V=800.0 PL=0
MOVL C00465 V=800.0 PL=0
MOVL C00466 V=800.0 PL=0
MOVL C00467 V=800.0 PL=0
MOVL C00468 V=800.0 PL=0
MOVL C00469 V=800.0 PL=0
MOVL C00470 V=800.0 PL=0
MOVL C00471 V=800.0 PL=0
MOVL C00472 V=800.0 PL=0
MOVL C00473 V=800.0 PL=0
MOVL C00474 V=800.0 PL=0
MOVL C00475 V=800.0 PL=0
MOVL C00476 V=800.0 PL=0
MOVL C00477 V=800.0 PL=0
MOVL C00478 V=800.0 PL=0
MOVL C00479 V=800.0 PL=0
MOVL C00480 V=800.0 PL=0
MOVL C00481 V=800.0 PL=0
MOVL C00482 V=800.0 PL=0
MOVL C00483 V=800.0 PL=0
MOVL C00484 V=800.0 PL=0
MOVL C00485 V=800.0 PL=0
MOVL C00486 V=800.0 PL=0
MOVL C00487 V=800.0 PL=0
MOVL C00488 V=800.0 PL=0
MOVL C00489 V=800.0 PL=0
MOVL C00490 V=800.0 PL=0
MOVL C00491 V=800.0 PL=0
MOVL C00492 V=800.0 PL=0
MOVL C00493 V=800.0 PL=0
MOVL C00494 V=800.0 PL=0
MOVL C00495 V=800.0 PL=0
MOVL C00496 V=800.0 PL=0
MOVL C00497 V=800.0 PL=0
MOVL C00498 V=800.0 PL=0
MOVL C00499 V=800.0 PL=0
MOVL C00500 V=800.0 PL=0
MOVL C00501 V=800.0 PL=0
MOVL C00502 V=800.0 PL=0
MOVL C00503 V=800.0 PL=0
MOVL C00504 V=800.0 PL=0
MOVL C00505 V=800.0 PL=0
MOVL C00506 V=800.0 PL=0
MOVL C00507 V=800.0 PL=0
MOVL C00508 V=800.0 PL=0
MOVL C00509 V=800.0 PL=0
MOVL C00510 V=800.0 PL=0
MOVL C00511 V=800.0 PL=0
MOVL C00512 V=800.0 PL=0
MOVL C00513 V=800.0 PL=0
MOVL C00514 V=800.0 PL=0
MOVL C00515 V=800.0 PL=0
MOVL C00516 V=800.0 PL=0
MOVL C00517 V=800.0 PL=0
MOVL C00518 V=800.0 PL=0
MOVL C00519 V=800.0 PL=0
MOVL C00520 V=800.0 PL=0
MOVL C00521 V=800.0 PL=0
MOVL C00522 V=800.0 PL=0
MOVL C00523 V=800.0 PL=0
MOVL C00524 V=800.0 PL=0
MOVL C00525 V=800.0 PL=0
MOVL C00526 V=800.0 PL=0
MOVL C00527 V=800.0 PL=0
MOVL C00528 V=800.0 PL=0
MOVL C00529 V=800.0 PL=0
MOVL C00530 V=800.0 PL=0
MOVL C00531 V=800.0 PL=0
MOVL C00532 V=800.0 PL=0
MOVL C00533 V=800.0 PL=0
MOVL C00534 V=800.0 PL=0
MOVL C00535 V=800.0 PL=0
MOVL C00536 V=800.0 PL=0
MOVL C00537 V=800.0 PL=0
MOVL C00538 V=800.0 PL=0
MOVL C00539 V=800.0 PL=0
MOVL C00540 V=800.0 PL=0
MOVL C00541 V=800.0 PL=0
MOVL C00542 V=800.0 PL=0
MOVL C00543 V=800.0 PL=0
MOVL C00544 V=800.0 PL=0
MOVL C00545 V=800.0 PL=0
MOVL C00546 V=800.0 PL=0
MOVL C00547 V=800.0 PL=0
MOVL C00548 V=800.0 PL=0
MOVL C00549 V=800.0 PL=0
MOVL C00550 V=800.0 PL=0
MOVL C00551 V=800.0 PL=0
MOVL C00552 V=800.0 PL=0
MOVL C00553 V=800.0 PL=0
MOVL C00554 V=800.0 PL=0
MOVL C00555 V=800.0 PL=0
MOVL C00556 V=800.0 PL=0
MOVL C00557 V=800.0 PL=0
MOVL C00558 V=800.0 PL=0
MOVL C00559 V=800.0 PL=0
MOVL C00560 V=800.0 PL=0
MOVL C00561 V=800.0 PL=0
MOVL C00562 V=800.0 PL=0
MOVL C00563 V=800.0 PL=0
MOVL C00564 V=800.0 PL=0
MOVL C00565 V=800.0 PL=0
MOVL C00566 V=800.0 PL=0
MOVL C00567 V=800.0 PL=0
MOVL C00568 V=800.0 PL=0
MOVL C00569 V=800.0 PL=0
MOVL C00570 V=800.0 PL=0
MOVL C00571 V=800.0 PL=0
MOVL C00572 V=800.0 PL=0
MOVL C00573 V=800.0 PL=0
MOVL C00574 V=800.0 PL=0
MOVL C00575 V=800.0 PL=0
MOVL C00576 V=800.0 PL=0
MOVL C00577 V=800.0 PL=0
MOVL C00578 V=800.0 PL=0
MOVL C00579 V=800.0 PL=0
MOVL C00580 V=800.0 PL=0
MOVL C00581 V=800.0 PL=0
MOVL C00582 V=800.0 PL=0
MOVL C00583 V=800.0 PL=0
MOVL C00584 V=800.0 PL=0
MOVL C00585 V=800.0 PL=0
MOVL C00586 V=800.0 PL=0
MOVL C00587 V=800.0 PL=0
MOVL C00588 V=800.0 PL=0
MOVL C00589 V=800.0 PL=0
MOVL C00590 V=800.0 PL=0
MOVL C00591 V=800.0 PL=0
MOVL C00592 V=800.0 PL=0
MOVL C00593 V=800.0 PL=0
MOVL C00594 V=800.0 PL=0
MOVL C00595 V=800.0 PL=0
MOVL C00596 V=800.0 PL=0
MOVL C00597 V=800.0 PL=0
MOVL C00598 V=800.0 PL=0
MOVL C00599 V=800.0 PL=0
MOVL C00600 V=800.0 PL=0
MOVL C00601 V=800.0 PL=0
MOVL C00602 V=800.0 PL=0
MOVL C00603 V=800.0 PL=0
MOVL C00604 V=800.0 PL=0
MOVL C00605 V=800.0 PL=0
MOVL C00606 V=800.0 PL=0
MOVL C00607 V=800.0 PL=0
MOVL C00608 V=800.0 PL=0
MOVL C00609 V=800.0 PL=0
MOVL C00610 V=800.0 PL=0
MOVL C00611 V=800.0 PL=0
MOVL C00612 V=800.0 PL=0
MOVL C00613 V=800.0 PL=0
MOVL C00614 V=800.0 PL=0
MOVL C00615 V=800.0 PL=0
MOVL C00616 V=800.0 PL=0
MOVL C00617 V=800.0 PL=0
MOVL C00618 V=800.0 PL=0
MOVL C00619 V=800.0 PL=0
MOVL C00620 V=800.0 PL=0
MOVL C00621 V=800.0 PL=0
MOVL C00622 V=800.0 PL=0
MOVL C00623 V=800.0 PL=0
MOVL C00624 V=800.0 PL=0
MOVL C00625 V=800.0 PL=0
MOVL C00626 V=800.0 PL=0
MOVL C00627 V=800.0 PL=0
MOVL C00628 V=800.0 PL=0
MOVL C00629 V=800.0 PL=0
MOVL C00630 V=800.0 PL=0
MOVL C00631 V=800.0 PL=0
MOVL C00632 V=800.0 PL=0
MOVL C00633 V=800.0 PL=0
MOVL C00634 V=800.0 PL=0
MOVL C00635 V=800.0 PL=0
MOVL C00636 V=800.0 PL=0
MOVL C00637 V=800.0 PL=0
MOVL C00638 V=800.0 PL=0
MOVL C00639 V=800.0 PL=0
MOVL C00640 V=800.0 PL=0
MOVL C00641 V=800.0 PL=0
MOVL C00642 V=800.0 PL=0
MOVL C00643 V=800.0 PL=0
MOVL C00644 V=800.0 PL=0
MOVL C00645 V=800.0 PL=0
MOVL C00646 V=800.0 PL=0
MOVL C00647 V=800.0 PL=0
MOVL C00648 V=800.0 PL=0
MOVL C00649 V=800.0 PL=0
MOVL C00650 V=800.0 PL=0
MOVL C00651 V=800.0 PL=0
MOVL C00652 V=800.0 PL=0
MOVL C00653 V=800.0 PL=0
MOVL C00654 V=800.0 PL=0
MOVL C00655 V=800.0 PL=0
MOVL C00656 V=800.0 PL=0
MOVL C00657 V=800.0 PL=0
MOVL C00658 V=800.0 PL=0
MOVL C00659 V=800.0 PL=0
MOVL C00660 V=800.0 PL=0
MOVL C00661 V=800.0 PL=0
MOVL C00662 V=800.0 PL=0
MOVL C00663 V=800.0 PL=0
MOVL C00664 V=800.0 PL=0
MOVL C00665 V=800.0 PL=0
MOVL C00666 V=800.0 PL=0
MOVL C00667 V=800.0 PL=0
MOVL C00668 V=800.0 PL=0
MOVL C00669 V=800.0 PL=0
MOVL C00670 V=800.0 PL=0
MOVL C00671 V=800.0 PL=0
MOVL C00672 V=800.0 PL=0
MOVL C00673 V=800.0 PL=0
MOVL C00674 V=800.0 PL=0
MOVL C00675 V=800.0 PL=0
MOVL C00676 V=800.0 PL=0
MOVL C00677 V=800.0 PL=0
MOVL C00678 V=800.0 PL=0
MOVL C00679 V=800.0 PL=0
MOVL C00680 V=800.0 PL=0
MOVL C00681 V=800.0 PL=0
MOVL C00682 V=800.0 PL=0
MOVL C00683 V=800.0 PL=0
MOVL C00684 V=800.0 PL=0
MOVL C00685 V=800.0 PL=0
MOVL C00686 V=800.0 PL=0
MOVL C00687 V=800.0 PL=0
MOVL C00688 V=800.0 PL=0
MOVL C00689 V=800.0 PL=0
MOVL C00690 V=800.0 PL=0
MOVL C00691 V=800.0 PL=0
MOVL C00692 V=800.0 PL=0
MOVL C00693 V=800.0 PL=0
MOVL C00694 V=800.0 PL=0
MOVL C00695 V=800.0 PL=0
MOVL C00696 V=800.0 PL=0
MOVL C00697 V=800.0 PL=0
MOVL C00698 V=800.0 PL=0
MOVL C00699 V=800.0 PL=0
MOVL C00700 V=800.0 PL=0
MOVL C00701 V=800.0 PL=0
MOVL C00702 V=800.0 PL=0
MOVL C00703 V=800.0 PL=0
MOVL C00704 V=800.0 PL=0
MOVL C00705 V=800.0 PL=0
MOVL C00706 V=800.0 PL=0
MOVL C00707 V=800.0 PL=0
MOVL C00708 V=800.0 PL=0
MOVL C00709 V=800.0 PL=0
MOVL C00710 V=800.0 PL=0
MOVL C00711 V=800.0 PL=0
MOVL C00712 V=800.0 PL=0
MOVL C00713 V=800.0 PL=0
MOVL C00714 V=800.0 PL=0
MOVL C00715 V=800.0 PL=0
MOVL C00716 V=800.0 PL=0
MOVL C00717 V=800.0 PL=0
MOVL C00718 V=800.0 PL=0
MOVL C00719 V=800.0 PL=0
MOVL C00720 V=800.0 PL=0
MOVL C00721 V=800.0 PL=0
MOVL C00722 V=800.0 PL=0
MOVL C00723 V=800.0 PL=0
MOVL C00724 V=800.0 PL=0
MOVL C00725 V=800.0 PL=0
MOVL C00726 V=800.0 PL=0
MOVL C00727 V=800.0 PL=0
MOVL C00728 V=800.0 PL=0
MOVL C00729 V=800.0 PL=0
MOVL C00730 V=800.0 PL=0
MOVL C00731 V=800.0 PL=0
MOVL C00732 V=800.0 PL=0
MOVL C00733 V=800.0 PL=0
MOVL C00734 V=800.0 PL=0
MOVL C00735 V=800.0 PL=0
MOVL C00736 V=800.0 PL=0
MOVL C00737 V=800.0 PL=0
MOVL C00738 V=800.0 PL=0
MOVL C00739 V=800.0 PL=0
MOVL C00740 V=800.0 PL=0
MOVL C00741 V=800.0 PL=0
MOVL C00742 V=800.0 PL=0
MOVL C00743 V=800.0 PL=0
MOVL C00744 V=800.0 PL=0
MOVL C00745 V=800.0 PL=0
MOVL C00746 V=800.0 PL=0
MOVL C00747 V=800.0 PL=0
MOVL C00748 V=800.0 PL=0
MOVL C00749 V=800.0 PL=0
MOVL C00750 V=800.0 PL=0
MOVL C00751 V=800.0 PL=0
MOVL C00752 V=800.0 PL=0
MOVL C00753 V=800.0 PL=0
MOVL C00754 V=800.0 PL=0
MOVL C00755 V=800.0 PL=0
MOVL C00756 V=800.0 PL=0
MOVL C00757 V=800.0 PL=0
MOVL C00758 V=800.0 PL=0
MOVL C00759 V=800.0 PL=0
MOVL C00760 V=800.0 PL=0
MOVL C00761 V=800.0 PL=0
MOVL C00762 V=800.0 PL=0
MOVL C00763 V=800.0 PL=0
MOVL C00764 V=800.0 PL=0
MOVL C00765 V=800.0 PL=0
MOVL C00766 V=800.0 PL=0
MOVL C00767 V=800.0 PL=0
MOVL C00768 V=800.0 PL=0
MOVL C00769 V=800.0 PL=0
MOVL C00770 V=800.0 PL=0
MOVL C00771 V=800.0 PL=0
MOVL C00772 V=800.0 PL=0
MOVL C00773 V=800.0 PL=0
MOVL C00774 V=800.0 PL=0
MOVL C00775 V=800.0 PL=0
MOVL C00776 V=800.0 PL=0
MOVL C00777 V=800.0 PL=0
MOVL C00778 V=800.0 PL=0
MOVL C00779 V=800.0 PL=0
MOVL C00780 V=800.0 PL=0
MOVL C00781 V=800.0 PL=0
MOVL C00782 V=800.0 PL=0
MOVL C00783 V=800.0 PL=0
MOVL C00784 V=800.0 PL=0
MOVL C00785 V=800.0 PL=0
MOVL C00786 V=800.0 PL=0
MOVL C00787 V=800.0 PL=0
MOVL C00788 V=800.0 PL=0
MOVL C00789 V=800.0 PL=0
MOVL C00790 V=800.0 PL=0
MOVL C00791 V=800.0 PL=0
MOVL C00792 V=800.0 PL=0
MOVL C00793 V=800.0 PL=0
MOVL C00794 V=800.0 PL=0
MOVL C00795 V=800.0 PL=0
MOVL C00796 V=800.0 PL=0
MOVL C00797 V=800.0 PL=0
MOVL C00798 V=800.0 PL=0
MOVL C00799 V=800.0 PL=0
MOVL C00800 V=800.0 PL=0
MOVL C00801 V=800.0 PL=0
MOVL C00802 V=800.0 PL=0
MOVL C00803 V=800.0 PL=0
MOVL C00804 V=800.0 PL=0
MOVL C00805 V=800.0 PL=0
MOVL C00806 V=800.0 PL=0
MOVL C00807 V=800.0 PL=0
MOVL C00808 V=800.0 PL=0
MOVL C00809 V=800.0 PL=0
MOVL C00810 V=800.0 PL=0
MOVL C00811 V=800.0 PL=0
MOVL C00812 V=800.0 PL=0
MOVL C00813 V=800.0 PL=0
MOVL C00814 V=800.0 PL=0
MOVL C00815 V=800.0 PL=0
MOVL C00816 V=800.0 PL=0
MOVL C00817 V=800.0 PL=0
MOVL C00818 V=800.0 PL=0
MOVL C00819 V=800.0 PL=0
MOVL C00820 V=800.0 PL=0
MOVL C00821 V=800.0 PL=0
MOVL C00822 V=800.0 PL=0
MOVL C00823 V=800.0 PL=0
MOVL C00824 V=800.0 PL=0
MOVL C00825 V=800.0 PL=0
MOVL C00826 V=800.0 PL=0
MOVL C00827 V=800.0 PL=0
MOVL C00828 V=800.0 PL=0
MOVL C00829 V=800.0 PL=0
MOVL C00830 V=800.0 PL=0
MOVL C00831 V=800.0 PL=0
MOVL C00832 V=800.0 PL=0
MOVL C00833 V=800.0 PL=0
MOVL C00834 V=800.0 PL=0
MOVL C00835 V=800.0 PL=0
MOVL C00836 V=800.0 PL=0
MOVL C00837 V=800.0 PL=0
MOVL C00838 V=800.0 PL=0
MOVL C00839 V=800.0 PL=0
MOVL C00840 V=800.0 PL=0
MOVL C00841 V=800.0 PL=0
MOVL C00842 V=800.0 PL=0
MOVL C00843 V=800.0 PL=0
MOVL C00844 V=800.0 PL=0
MOVL C00845 V=800.0 PL=0
MOVL C00846 V=800.0 PL=0
MOVL C00847 V=800.0 PL=0
MOVL C00848 V=800.0 PL=0
MOVL C00849 V=800.0 PL=0
MOVL C00850 V=800.0 PL=0
MOVL C00851 V=800.0 PL=0
MOVL C00852 V=800.0 PL=0
MOVL C00853 V=800.0 PL=0
MOVL C00854 V=800.0 PL=0
MOVL C00855 V=800.0 PL=0
MOVL C00856 V=800.0 PL=0
MOVL C00857 V=800.0 PL=0
MOVL C00858 V=800.0 PL=0
MOVL C00859 V=800.0 PL=0
MOVL C00860 V=800.0 PL=0
MOVL C00861 V=800.0 PL=0
MOVL C00862 V=800.0 PL=0
MOVL C00863 V=800.0 PL=0
MOVL C00864 V=800.0 PL=0
MOVL C00865 V=800.0 PL=0
MOVL C00866 V=800.0 PL=0
MOVL C00867 V=800.0 PL=0
MOVL C00868 V=800.0 PL=0
MOVL C00869 V=800.0 PL=0
MOVL C00870 V=800.0 PL=0
MOVL C00871 V=800.0 PL=0
MOVL C00872 V=800.0 PL=0
MOVL C00873 V=800.0 PL=0
MOVL C00874 V=800.0 PL=0
MOVL C00875 V=800.0 PL=0
MOVL C00876 V=800.0 PL=0
MOVL C00877 V=800.0 PL=0
MOVL C00878 V=800.0 PL=0
MOVL C00879 V=800.0 PL=0
MOVL C00880 V=800.0 PL=0
MOVL C00881 V=800.0 PL=0
MOVL C00882 V=800.0 PL=0
MOVL C00883 V=800.0 PL=0
MOVL C00884 V=800.0 PL=0
MOVL C00885 V=800.0 PL=0
MOVL C00886 V=800.0 PL=0
MOVL C00887 V=800.0 PL=0
MOVL C00888 V=800.0 PL=0
MOVL C00889 V=800.0 PL=0
MOVL C00890 V=800.0 PL=0
MOVL C00891 V=800.0 PL=0
MOVL C00892 V=800.0 PL=0
MOVL C00893 V=800.0 PL=0
MOVL C00894 V=800.0 PL=0
MOVL C00895 V=800.0 PL=0
MOVL C00896 V=800.0 PL=0
MOVL C00897 V=800.0 PL=0
MOVL C00898 V=800.0 PL=0
MOVL C00899 V=800.0 PL=0
MOVL C00900 V=800.0 PL=0
MOVL C00901 V=800.0 PL=0
MOVL C00902 V=800.0 PL=0
MOVL C00903 V=800.0 PL=0
MOVL C00904 V=800.0 PL=0
MOVL C00905 V=800.0 PL=0
MOVL C00906 V=800.0 PL=0
MOVL C00907 V=800.0 PL=0
MOVL C00908 V=800.0 PL=0
MOVL C00909 V=800.0 PL=0
MOVL C00910 V=800.0 PL=0
MOVL C00911 V=800.0 PL=0
MOVL C00912 V=800.0 PL=0
MOVL C00913 V=800.0 PL=0
MOVL C00914 V=800.0 PL=0
MOVL C00915 V=800.0 PL=0
MOVL C00916 V=800.0 PL=0
MOVL C00917 V=800.0 PL=0
MOVL C00918 V=800.0 PL=0
MOVL C00919 V=800.0 PL=0
MOVL C00920 V=800.0 PL=0
MOVL C00921 V=800.0 PL=0
MOVL C00922 V=800.0 PL=0
MOVL C00923 V=800.0 PL=0
MOVL C00924 V=800.0 PL=0
MOVL C00925 V=800.0 PL=0
MOVL C00926 V=800.0 PL=0
MOVL C00927 V=800.0 PL=0
MOVL C00928 V=800.0 PL=0
MOVL C00929 V=800.0 PL=0
MOVL C00930 V=800.0 PL=0
MOVL C00931 V=800.0 PL=0
MOVL C00932 V=800.0 PL=0
MOVL C00933 V=800.0 PL=0
MOVL C00934 V=800.0 PL=0
MOVL C00935 V=800.0 PL=0
MOVL C00936 V=800.0 PL=0
MOVL C00937 V=800.0 PL=0
MOVL C00938 V=800.0 PL=0
MOVL C00939 V=800.0 PL=0
MOVL C00940 V=800.0 PL=0
MOVL C00941 V=800.0 PL=0
MOVL C00942 V=800.0 PL=0
MOVL C00943 V=800.0 PL=0
MOVL C00944 V=800.0 PL=0
MOVL C00945 V=800.0 PL=0
MOVL C00946 V=800.0 PL=0
MOVL C00947 V=800.0 PL=0
MOVL C00948 V=800.0 PL=0
MOVL C00949 V=800.0 PL=0
MOVL C00950 V=800.0 PL=0
MOVL C00951 V=800.0 PL=0
MOVL C00952 V=800.0 PL=0
MOVL C00953 V=800.0 PL=0
MOVL C00954 V=800.0 PL=0
MOVL C00955 V=800.0 PL=0
MOVL C00956 V=800.0 PL=0
MOVL C00957 V=800.0 PL=0
MOVL C00958 V=800.0 PL=0
MOVL C00959 V=800.0 PL=0
MOVL C00960 V=800.0 PL=0
MOVL C00961 V=800.0 PL=0
MOVL C00962 V=800.0 PL=0
MOVL C00963 V=800.0 PL=0
MOVL C00964 V=800.0 PL=0
MOVL C00965 V=800.0 PL=0
MOVL C00966 V=800.0 PL=0
MOVL C00967 V=800.0 PL=0
MOVL C00968 V=800.0 PL=0
MOVL C00969 V=800.0 PL=0
MOVL C00970 V=800.0 PL=0
MOVL C00971 V=800.0 PL=0
MOVL C00972 V=800.0 PL=0
MOVL C00973 V=800.0 PL=0
MOVL C00974 V=800.0 PL=0
MOVL C00975 V=800.0 PL=0
MOVL C00976 V=800.0 PL=0
MOVL C00977 V=800.0 PL=0
MOVL C00978 V=800.0 PL=0
MOVL C00979 V=800.0 PL=0
MOVL C00980 V=800.0 PL=0
MOVL C00981 V=800.0 PL=0
MOVL C00982 V=800.0 PL=0
MOVL C00983 V=800.0 PL=0
MOVL C00984 V=800.0 PL=0
MOVL C00985 V=800.0 PL=0
MOVL C00986 V=800.0 PL=0
MOVL C00987 V=800.0 PL=0
MOVL C00988 V=800.0 PL=0
MOVL C00989 V=800.0 PL=0
MOVL C00990 V=800.0 PL=0
MOVL C00991 V=800.0 PL=0
MOVL C00992 V=800.0 PL=0
MOVL C00993 V=800.0 PL=0
MOVL C00994 V=800.0 PL=0
MOVL C00995 V=800.0 PL=0
MOVL C00996 V=800.0 PL=0
MOVL C00997 V=800.0 PL=0
MOVL C00998 V=800.0 PL=0
MOVL C00999 V=800.0 PL=0
MOVL C01000 V=800.0 PL=0
MOVL C01001 V=800.0 PL=0
MOVL C01002 V=800.0 PL=0
MOVL C01003 V=800.0 PL=0
MOVL C01004 V=800.0 PL=0
MOVL C01005 V=800.0 PL=0
MOVL C01006 V=800.0 PL=0
MOVL C01007 V=800.0 PL=0
MOVL C01008 V=800.0 PL=0
MOVL C01009 V=800.0 PL=0
MOVL C01010 V=800.0 PL=0
MOVL C01011 V=800.0 PL=0
MOVL C01012 V=800.0 PL=0
MOVL C01013 V=800.0 PL=0
MOVL C01014 V=800.0 PL=0
MOVL C01015 V=800.0 PL=0
MOVL C01016 V=800.0 PL=0
MOVL C01017 V=800.0 PL=0
MOVL C01018 V=800.0 PL=0
MOVL C01019 V=800.0 PL=0
MOVL C01020 V=800.0 PL=0
MOVL C01021 V=800.0 PL=0
MOVL C01022 V=800.0 PL=0
MOVL C01023 V=800.0 PL=0
MOVL C01024 V=800.0 PL=0
MOVL C01025 V=800.0 PL=0
MOVL C01026 V=800.0 PL=0
MOVL C01027 V=800.0 PL=0
MOVL C01028 V=800.0 PL=0
MOVL C01029 V=800.0 PL=0
MOVL C01030 V=800.0 PL=0
MOVL C01031 V=800.0 PL=0
MOVL C01032 V=800.0 PL=0
MOVL C01033 V=800.0 PL=0
MOVL C01034 V=800.0 PL=0
MOVL C01035 V=800.0 PL=0
MOVL C01036 V=800.0 PL=0
MOVL C01037 V=800.0 PL=0
MOVL C01038 V=800.0 PL=0
MOVL C01039 V=800.0 PL=0
MOVL C01040 V=800.0 PL=0
MOVL C01041 V=800.0 PL=0
MOVL C01042 V=800.0 PL=0
MOVL C01043 V=800.0 PL=0
MOVL C01044 V=800.0 PL=0
MOVL C01045 V=800.0 PL=0
MOVL C01046 V=800.0 PL=0
MOVL C01047 V=800.0 PL=0
MOVL C01048 V=800.0 PL=0
MOVL C01049 V=800.0 PL=0
MOVL C01050 V=800.0 PL=0
MOVL C01051 V=800.0 PL=0
MOVL C01052 V=800.0 PL=0
MOVL C01053 V=800.0 PL=0
MOVL C01054 V=800.0 PL=0
MOVL C01055 V=800.0 PL=0
MOVL C01056 V=800.0 PL=0
MOVL C01057 V=800.0 PL=0
MOVL C01058 V=800.0 PL=0
MOVL C01059 V=800.0 PL=0
MOVL C01060 V=800.0 PL=0
MOVL C01061 V=800.0 PL=0
MOVL C01062 V=800.0 PL=0
MOVL C01063 V=800.0 PL=0
MOVL C01064 V=800.0 PL=0
MOVL C01065 V=800.0 PL=0
MOVL C01066 V=800.0 PL=0
MOVL C01067 V=800.0 PL=0
MOVL C01068 V=800.0 PL=0
MOVL C01069 V=800.0 PL=0
MOVL C01070 V=800.0 PL=0
MOVL C01071 V=800.0 PL=0
MOVL C01072 V=800.0 PL=0
MOVL C01073 V=800.0 PL=0
MOVL C01074 V=800.0 PL=0
MOVL C01075 V=800.0 PL=0
MOVL C01076 V=800.0 PL=0
MOVL C01077 V=800.0 PL=0
MOVL C01078 V=800.0 PL=0
MOVL C01079 V=800.0 PL=0
MOVL C01080 V=800.0 PL=0
MOVL C01081 V=800.0 PL=0
MOVL C01082 V=800.0 PL=0
MOVL C01083 V=800.0 PL=0
MOVL C01084 V=800.0 PL=0
MOVL C01085 V=800.0 PL=0
MOVL C01086 V=800.0 PL=0
MOVL C01087 V=800.0 PL=0
MOVL C01088 V=800.0 PL=0
MOVL C01089 V=800.0 PL=0
MOVL C01090 V=800.0 PL=0
MOVL C01091 V=800.0 PL=0
MOVL C01092 V=800.0 PL=0
MOVL C01093 V=800.0 PL=0
MOVL C01094 V=800.0 PL=0
MOVL C01095 V=800.0 PL=0
MOVL C01096 V=800.0 PL=0
MOVL C01097 V=800.0 PL=0
MOVL C01098 V=800.0 PL=0
MOVL C01099 V=800.0 PL=0
MOVL C01100 V=800.0 PL=0
MOVL C01101 V=800.0 PL=0
MOVL C01102 V=800.0 PL=0
MOVL C01103 V=800.0 PL=0
MOVL C01104 V=800.0 PL=0
MOVL C01105 V=800.0 PL=0
MOVL C01106 V=800.0 PL=0
MOVL C01107 V=800.0 PL=0
MOVL C01108 V=800.0 PL=0
MOVL C01109 V=800.0 PL=0
MOVL C01110 V=800.0 PL=0
MOVL C01111 V=800.0 PL=0
MOVL C01112 V=800.0 PL=0
MOVL C01113 V=800.0 PL=0
MOVL C01114 V=800.0 PL=0
MOVL C01115 V=800.0 PL=0
MOVL C01116 V=800.0 PL=0
MOVL C01117 V=800.0 PL=0
MOVL C01118 V=800.0 PL=0
MOVL C01119 V=800.0 PL=0
MOVL C01120 V=800.0 PL=0
MOVL C01121 V=800.0 PL=0
MOVL C01122 V=800.0 PL=0
MOVL C01123 V=800.0 PL=0
MOVL C01124 V=800.0 PL=0
MOVL C01125 V=800.0 PL=0
MOVL C01126 V=800.0 PL=0
MOVL C01127 V=800.0 PL=0
MOVL C01128 V=800.0 PL=0
MOVL C01129 V=800.0 PL=0
MOVL C01130 V=800.0 PL=0
MOVL C01131 V=800.0 PL=0
MOVL C01132 V=800.0 PL=0
MOVL C01133 V=800.0 PL=0
MOVL C01134 V=800.0 PL=0
MOVL C01135 V=800.0 PL=0
MOVL C01136 V=800.0 PL=0
MOVL C01137 V=800.0 PL=0
MOVL C01138 V=800.0 PL=0
MOVL C01139 V=800.0 PL=0
MOVL C01140 V=800.0 PL=0
MOVL C01141 V=800.0 PL=0
MOVL C01142 V=800.0 PL=0
MOVL C01143 V=800.0 PL=0
MOVL C01144 V=800.0 PL=0
MOVL C01145 V=800.0 PL=0
MOVL C01146 V=800.0 PL=0
MOVL C01147 V=800.0 PL=0
MOVL C01148 V=800.0 PL=0
MOVL C01149 V=800.0 PL=0
MOVL C01150 V=800.0 PL=0
MOVL C01151 V=800.0 PL=0
MOVL C01152 V=800.0 PL=0
MOVL C01153 V=800.0 PL=0
MOVL C01154 V=800.0 PL=0
MOVL C01155 V=800.0 PL=0
MOVL C01156 V=800.0 PL=0
MOVL C01157 V=800.0 PL=0
MOVL C01158 V=800.0 PL=0
MOVL C01159 V=800.0 PL=0
MOVL C01160 V=800.0 PL=0
MOVL C01161 V=800.0 PL=0
MOVL C01162 V=800.0 PL=0
MOVL C01163 V=800.0 PL=0
MOVL C01164 V=800.0 PL=0
MOVL C01165 V=800.0 PL=0
MOVL C01166 V=800.0 PL=0
MOVL C01167 V=800.0 PL=0
MOVL C01168 V=800.0 PL=0
MOVL C01169 V=800.0 PL=0
MOVL C01170 V=800.0 PL=0
MOVL C01171 V=800.0 PL=0
MOVL C01172 V=800.0 PL=0
MOVL C01173 V=800.0 PL=0
MOVL C01174 V=800.0 PL=0
MOVL C01175 V=800.0 PL=0
MOVL C01176 V=800.0 PL=0
MOVL C01177 V=800.0 PL=0
MOVL C01178 V=800.0 PL=0
MOVL C01179 V=800.0 PL=0
MOVL C01180 V=800.0 PL=0
MOVL C01181 V=800.0 PL=0
MOVL C01182 V=800.0 PL=0
MOVL C01183 V=800.0 PL=0
MOVL C01184 V=800.0 PL=0
MOVL C01185 V=800.0 PL=0
MOVL C01186 V=800.0 PL=0
MOVL C01187 V=800.0 PL=0
MOVL C01188 V=800.0 PL=0
MOVL C01189 V=800.0 PL=0
MOVL C01190 V=800.0 PL=0
MOVL C01191 V=800.0 PL=0
MOVL C01192 V=800.0 PL=0
MOVL C01193 V=800.0 PL=0
MOVL C01194 V=800.0 PL=0
MOVL C01195 V=800.0 PL=0
MOVL C01196 V=800.0 PL=0
MOVL C01197 V=800.0 PL=0
MOVL C01198 V=800.0 PL=0
MOVL C01199 V=800.0 PL=0
MOVL C01200 V=800.0 PL=0
MOVL C01201 V=800.0 PL=0
MOVL C01202 V=800.0 PL=0
MOVL C01203 V=800.0 PL=0
MOVL C01204 V=800.0 PL=0
MOVL C01205 V=800.0 PL=0
MOVL C01206 V=800.0 PL=0
MOVL C01207 V=800.0 PL=0
MOVL C01208 V=800.0 PL=0
MOVL C01209 V=800.0 PL=0
MOVL C01210 V=800.0 PL=0
MOVL C01211 V=800.0 PL=0
MOVL C01212 V=800.0 PL=0
MOVL C01213 V=800.0 PL=0
MOVL C01214 V=800.0 PL=0
MOVL C01215 V=800.0 PL=0
MOVL C01216 V=800.0 PL=0
MOVL C01217 V=800.0 PL=0
MOVL C01218 V=800.0 PL=0
MOVL C01219 V=800.0 PL=0
MOVL C01220 V=800.0 PL=0
MOVL C01221 V=800.0 PL=0
MOVL C01222 V=800.0 PL=0
MOVL C01223 V=800.0 PL=0
MOVL C01224 V=800.0 PL=0
MOVL C01225 V=800.0 PL=0
MOVL C01226 V=800.0 PL=0
MOVL C01227 V=800.0 PL=0
MOVL C01228 V=800.0 PL=0
MOVL C01229 V=800.0 PL=0
MOVL C01230 V=800.0 PL=0
MOVL C01231 V=800.0 PL=0
MOVL C01232 V=800.0 PL=0
MOVL C01233 V=800.0 PL=0
MOVL C01234 V=800.0 PL=0
MOVL C01235 V=800.0 PL=0
MOVL C01236 V=800.0 PL=0
MOVL C01237 V=800.0 PL=0
MOVL C01238 V=800.0 PL=0
MOVL C01239 V=800.0 PL=0
MOVL C01240 V=800.0 PL=0
MOVL C01241 V=800.0 PL=0
MOVL C01242 V=800.0 PL=0
MOVL C01243 V=800.0 PL=0
MOVL C01244 V=800.0 PL=0
MOVL C01245 V=800.0 PL=0
MOVL C01246 V=800.0 PL=0
MOVL C01247 V=800.0 PL=0
MOVL C01248 V=800.0 PL=0
MOVL C01249 V=800.0 PL=0
MOVL C01250 V=800.0 PL=0
MOVL C01251 V=800.0 PL=0
MOVL C01252 V=800.0 PL=0
MOVL C01253 V=800.0 PL=0
MOVL C01254 V=800.0 PL=0
MOVL C01255 V=800.0 PL=0
MOVL C01256 V=800.0 PL=0
MOVL C01257 V=800.0 PL=0
MOVL C01258 V=800.0 PL=0
MOVL C01259 V=800.0 PL=0
MOVL C01260 V=800.0 PL=0
MOVL C01261 V=800.0 PL=0
MOVL C01262 V=800.0 PL=0
MOVL C01263 V=800.0 PL=0
MOVL C01264 V=800.0 PL=0
MOVL C01265 V=800.0 PL=0
MOVL C01266 V=800.0 PL=0
MOVL C01267 V=800.0 PL=0
MOVL C01268 V=800.0 PL=0
MOVL C01269 V=800.0 PL=0
MOVL C01270 V=800.0 PL=0
MOVL C01271 V=800.0 PL=0
MOVL C01272 V=800.0 PL=0
MOVL C01273 V=800.0 PL=0
MOVL C01274 V=800.0 PL=0
MOVL C01275 V=800.0 PL=0
MOVL C01276 V=800.0 PL=0
MOVL C01277 V=800.0 PL=0
MOVL C01278 V=800.0 PL=0
MOVL C01279 V=800.0 PL=0
MOVL C01280 V=800.0 PL=0
MOVL C01281 V=800.0 PL=0
MOVL C01282 V=800.0 PL=0
MOVL C01283 V=800.0 PL=0
MOVL C01284 V=800.0 PL=0
MOVL C01285 V=800.0 PL=0
MOVL C01286 V=800.0 PL=0
MOVL C01287 V=800.0 PL=0
MOVL C01288 V=800.0 PL=0
MOVL C01289 V=800.0 PL=0
MOVL C01290 V=800.0 PL=0
MOVL C01291 V=800.0 PL=0
MOVL C01292 V=800.0 PL=0
MOVL C01293 V=800.0 PL=0
MOVL C01294 V=800.0 PL=0
MOVL C01295 V=800.0 PL=0
MOVL C01296 V=800.0 PL=0
MOVL C01297 V=800.0 PL=0
MOVL C01298 V=800.0 PL=0
MOVL C01299 V=800.0 PL=0
MOVL C01300 V=800.0 PL=0
MOVL C01301 V=800.0 PL=0
MOVL C01302 V=800.0 PL=0
MOVL C01303 V=800.0 PL=0
MOVL C01304 V=800.0 PL=0
MOVL C01305 V=800.0 PL=0
MOVL C01306 V=800.0 PL=0
MOVL C01307 V=800.0 PL=0
MOVL C01308 V=800.0 PL=0
MOVL C01309 V=800.0 PL=0
MOVL C01310 V=800.0 PL=0
MOVL C01311 V=800.0 PL=0
MOVL C01312 V=800.0 PL=0
MOVL C01313 V=800.0 PL=0
MOVL C01314 V=800.0 PL=0
MOVL C01315 V=800.0 PL=0
MOVL C01316 V=800.0 PL=0
MOVL C01317 V=800.0 PL=0
MOVL C01318 V=800.0 PL=0
MOVL C01319 V=800.0 PL=0
MOVL C01320 V=800.0 PL=0
MOVL C01321 V=800.0 PL=0
MOVL C01322 V=800.0 PL=0
MOVL C01323 V=800.0 PL=0
MOVL C01324 V=800.0 PL=0
MOVL C01325 V=800.0 PL=0
MOVL C01326 V=800.0 PL=0
MOVL C01327 V=800.0 PL=0
MOVL C01328 V=800.0 PL=0
MOVL C01329 V=800.0 PL=0
MOVL C01330 V=800.0 PL=0
MOVL C01331 V=800.0 PL=0
MOVL C01332 V=800.0 PL=0
MOVL C01333 V=800.0 PL=0
MOVL C01334 V=800.0 PL=0
MOVL C01335 V=800.0 PL=0
MOVL C01336 V=800.0 PL=0
MOVL C01337 V=800.0 PL=0
MOVL C01338 V=800.0 PL=0
MOVL C01339 V=800.0 PL=0
MOVL C01340 V=800.0 PL=0
MOVL C01341 V=800.0 PL=0
MOVL C01342 V=800.0 PL=0
MOVL C01343 V=800.0 PL=0
MOVL C01344 V=800.0 PL=0
MOVL C01345 V=800.0 PL=0
MOVL C01346 V=800.0 PL=0
MOVL C01347 V=800.0 PL=0
MOVL C01348 V=800.0 PL=0
MOVL C01349 V=800.0 PL=0
MOVL C01350 V=800.0 PL=0
MOVL C01351 V=800.0 PL=0
MOVL C01352 V=800.0 PL=0
MOVL C01353 V=800.0 PL=0
MOVL C01354 V=800.0 PL=0
MOVL C01355 V=800.0 PL=0
MOVL C01356 V=800.0 PL=0
MOVL C01357 V=800.0 PL=0
MOVL C01358 V=800.0 PL=0
MOVL C01359 V=800.0 PL=0
MOVL C01360 V=800.0 PL=0
MOVL C01361 V=800.0 PL=0
MOVL C01362 V=800.0 PL=0
MOVL C01363 V=800.0 PL=0
MOVL C01364 V=800.0 PL=0
MOVL C01365 V=800.0 PL=0
MOVL C01366 V=800.0 PL=0
MOVL C01367 V=800.0 PL=0
MOVL C01368 V=800.0 PL=0
MOVL C01369 V=800.0 PL=0
MOVL C01370 V=800.0 PL=0
MOVL C01371 V=800.0 PL=0
MOVL C01372 V=800.0 PL=0
MOVL C01373 V=800.0 PL=0
MOVL C01374 V=800.0 PL=0
MOVL C01375 V=800.0 PL=0
MOVL C01376 V=800.0 PL=0
MOVL C01377 V=800.0 PL=0
MOVL C01378 V=800.0 PL=0
MOVL C01379 V=800.0 PL=0
MOVL C01380 V=800.0 PL=0
MOVL C01381 V=800.0 PL=0
MOVL C01382 V=800.0 PL=0
MOVL C01383 V=800.0 PL=0
MOVL C01384 V=800.0 PL=0
MOVL C01385 V=800.0 PL=0
MOVL C01386 V=800.0 PL=0
MOVL C01387 V=800.0 PL=0
MOVL C01388 V=800.0 PL=0
MOVL C01389 V=800.0 PL=0
MOVL C01390 V=800.0 PL=0
MOVL C01391 V=800.0 PL=0
MOVL C01392 V=800.0 PL=0
MOVL C01393 V=800.0 PL=0
MOVL C01394 V=800.0 PL=0
MOVL C01395 V=800.0 PL=0
MOVL C01396 V=800.0 PL=0
MOVL C01397 V=800.0 PL=0
MOVL C01398 V=800.0 PL=0
MOVL C01399 V=800.0 PL=0
MOVL C01400 V=800.0 PL=0
MOVL C01401 V=800.0 PL=0
MOVL C01402 V=800.0 PL=0
MOVL C01403 V=800.0 PL=0
MOVL C01404 V=800.0 PL=0
MOVL C01405 V=800.0 PL=0
MOVL C01406 V=800.0 PL=0
MOVL C01407 V=800.0 PL=0
MOVL C01408 V=800.0 PL=0
MOVL C01409 V=800.0 PL=0
MOVL C01410 V=800.0 PL=0
MOVL C01411 V=800.0 PL=0
MOVL C01412 V=800.0 PL=0
MOVL C01413 V=800.0 PL=0
MOVL C01414 V=800.0 PL=0
MOVL C01415 V=800.0 PL=0
MOVL C01416 V=800.0 PL=0
MOVL C01417 V=800.0 PL=0
MOVL C01418 V=800.0 PL=0
MOVL C01419 V=800.0 PL=0
MOVL C01420 V=800.0 PL=0
MOVL C01421 V=800.0 PL=0
MOVL C01422 V=800.0 PL=0
MOVL C01423 V=800.0 PL=0
MOVL C01424 V=800.0 PL=0
MOVL C01425 V=800.0 PL=0
MOVL C01426 V=800.0 PL=0
MOVL C01427 V=800.0 PL=0
MOVL C01428 V=800.0 PL=0
MOVL C01429 V=800.0 PL=0
MOVL C01430 V=800.0 PL=0
MOVL C01431 V=800.0 PL=0
MOVL C01432 V=800.0 PL=0
MOVL C01433 V=800.0 PL=0
MOVL C01434 V=800.0 PL=0
MOVL C01435 V=800.0 PL=0
MOVL C01436 V=800.0 PL=0
MOVL C01437 V=800.0 PL=0
MOVL C01438 V=800.0 PL=0
MOVL C01439 V=800.0 PL=0
MOVL C01440 V=800.0 PL=0
MOVL C01441 V=800.0 PL=0
MOVL C01442 V=800.0 PL=0
MOVL C01443 V=800.0 PL=0
MOVL C01444 V=800.0 PL=0
MOVL C01445 V=800.0 PL=0
MOVL C01446 V=800.0 PL=0
MOVL C01447 V=800.0 PL=0
MOVL C01448 V=800.0 PL=0
MOVL C01449 V=800.0 PL=0
MOVL C01450 V=800.0 PL=0
MOVL C01451 V=800.0 PL=0
MOVL C01452 V=800.0 PL=0
MOVL C01453 V=800.0 PL=0
MOVL C01454 V=800.0 PL=0
MOVL C01455 V=800.0 PL=0
MOVL C01456 V=800.0 PL=0
MOVL C01457 V=800.0 PL=0
MOVL C01458 V=800.0 PL=0
MOVL C01459 V=800.0 PL=0
MOVL C01460 V=800.0 PL=0
MOVL C01461 V=800.0 PL=0
MOVL C01462 V=800.0 PL=0
MOVL C01463 V=800.0 PL=0
MOVL C01464 V=800.0 PL=0
MOVL C01465 V=800.0 PL=0
MOVL C01466 V=800.0 PL=0
MOVL C01467 V=800.0 PL=0
MOVL C01468 V=800.0 PL=0
MOVL C01469 V=800.0 PL=0
MOVL C01470 V=800.0 PL=0
MOVL C01471 V=800.0 PL=0
MOVL C01472 V=800.0 PL=0
MOVL C01473 V=800.0 PL=0
MOVL C01474 V=800.0 PL=0
MOVL C01475 V=800.0 PL=0
MOVL C01476 V=800.0 PL=0
MOVL C01477 V=800.0 PL=0
MOVL C01478 V=800.0 PL=0
MOVL C01479 V=800.0 PL=0
MOVL C01480 V=800.0 PL=0
MOVL C01481 V=800.0 PL=0
MOVL C01482 V=800.0 PL=0
MOVL C01483 V=800.0 PL=0
MOVL C01484 V=800.0 PL=0
MOVL C01485 V=800.0 PL=0
MOVL C01486 V=800.0 PL=0
MOVL C01487 V=800.0 PL=0
MOVL C01488 V=800.0 PL=0
MOVL C01489 V=800.0 PL=0
MOVL C01490 V=800.0 PL=0
MOVL C01491 V=800.0 PL=0
MOVL C01492 V=800.0 PL=0
MOVL C01493 V=800.0 PL=0
MOVL C01494 V=800.0 PL=0
MOVL C01495 V=800.0 PL=0
MOVL C01496 V=800.0 PL=0
MOVL C01497 V=800.0 PL=0
MOVL C01498 V=800.0 PL=0
MOVL C01499 V=800.0 PL=0
MOVL C01500 V=800.0 PL=0
MOVL C01501 V=800.0 PL=0
MOVL C01502 V=800.0 PL=0
MOVL C01503 V=800.0 PL=0
MOVL C01504 V=800.0 PL=0
MOVL C01505 V=800.0 PL=0
MOVL C01506 V=800.0 PL=0
MOVL C01507 V=800.0 PL=0
MOVL C01508 V=800.0 PL=0
MOVL C01509 V=800.0 PL=0
MOVL C01510 V=800.0 PL=0
MOVL C01511 V=800.0 PL=0
MOVL C01512 V=800.0 PL=0
MOVL C01513 V=800.0 PL=0
MOVL C01514 V=800.0 PL=0
MOVL C01515 V=800.0 PL=0
MOVL C01516 V=800.0 PL=0
MOVL C01517 V=800.0 PL=0
MOVL C01518 V=800.0 PL=0
MOVL C01519 V=800.0 PL=0
MOVL C01520 V=800.0 PL=0
MOVL C01521 V=800.0 PL=0
MOVL C01522 V=800.0 PL=0
MOVL C01523 V=800.0 PL=0
MOVL C01524 V=800.0 PL=0
MOVL C01525 V=800.0 PL=0
MOVL C01526 V=800.0 PL=0
MOVL C01527 V=800.0 PL=0
MOVL C01528 V=800.0 PL=0
MOVL C01529 V=800.0 PL=0
MOVL C01530 V=800.0 PL=0
MOVL C01531 V=800.0 PL=0
MOVL C01532 V=800.0 PL=0
MOVL C01533 V=800.0 PL=0
MOVL C01534 V=800.0 PL=0
MOVL C01535 V=800.0 PL=0
MOVL C01536 V=800.0 PL=0
MOVL C01537 V=800.0 PL=0
MOVL C01538 V=800.0 PL=0
MOVL C01539 V=800.0 PL=0
MOVL C01540 V=800.0 PL=0
MOVL C01541 V=800.0 PL=0
MOVL C01542 V=800.0 PL=0
MOVL C01543 V=800.0 PL=0
MOVL C01544 V=800.0 PL=0
MOVL C01545 V=800.0 PL=0
MOVL C01546 V=800.0 PL=0
MOVL C01547 V=800.0 PL=0
MOVL C01548 V=800.0 PL=0
MOVL C01549 V=800.0 PL=0
MOVL C01550 V=800.0 PL=0
MOVL C01551 V=800.0 PL=0
MOVL C01552 V=800.0 PL=0
MOVL C01553 V=800.0 PL=0
MOVL C01554 V=800.0 PL=0
MOVL C01555 V=800.0 PL=0
MOVL C01556 V=800.0 PL=0
MOVL C01557 V=800.0 PL=0
MOVL C01558 V=800.0 PL=0
MOVL C01559 V=800.0 PL=0
MOVL C01560 V=800.0 PL=0
MOVL C01561 V=800.0 PL=0
MOVL C01562 V=800.0 PL=0
MOVL C01563 V=800.0 PL=0
MOVL C01564 V=800.0 PL=0
MOVL C01565 V=800.0 PL=0
MOVL C01566 V=800.0 PL=0
MOVL C01567 V=800.0 PL=0
MOVL C01568 V=800.0 PL=0
MOVL C01569 V=800.0 PL=0
MOVL C01570 V=800.0 PL=0
MOVL C01571 V=800.0 PL=0
MOVL C01572 V=800.0 PL=0
MOVL C01573 V=800.0 PL=0
MOVL C01574 V=800.0 PL=0
MOVL C01575 V=800.0 PL=0
MOVL C01576 V=800.0 PL=0
MOVL C01577 V=800.0 PL=0
MOVL C01578 V=800.0 PL=0
MOVL C01579 V=800.0 PL=0
MOVL C01580 V=800.0 PL=0
MOVL C01581 V=800.0 PL=0
MOVL C01582 V=800.0 PL=0
MOVL C01583 V=800.0 PL=0
MOVL C01584 V=800.0 PL=0
MOVL C01585 V=800.0 PL=0
MOVL C01586 V=800.0 PL=0
MOVL C01587 V=800.0 PL=0
MOVL C01588 V=800.0 PL=0
MOVL C01589 V=800.0 PL=0
MOVL C01590 V=800.0 PL=0
MOVL C01591 V=800.0 PL=0
MOVL C01592 V=800.0 PL=0
MOVL C01593 V=800.0 PL=0
MOVL C01594 V=800.0 PL=0
MOVL C01595 V=800.0 PL=0
MOVL C01596 V=800.0 PL=0
MOVL C01597 V=800.0 PL=0
MOVL C01598 V=800.0 PL=0
MOVL C01599 V=800.0 PL=0
MOVL C01600 V=800.0 PL=0
MOVL C01601 V=800.0 PL=0
MOVL C01602 V=800.0 PL=0
MOVL C01603 V=800.0 PL=0
MOVL C01604 V=800.0 PL=0
MOVL C01605 V=800.0 PL=0
MOVL C01606 V=800.0 PL=0
MOVL C01607 V=800.0 PL=0
MOVL C01608 V=800.0 PL=0
MOVL C01609 V=800.0 PL=0
MOVL C01610 V=800.0 PL=0
MOVL C01611 V=800.0 PL=0
MOVL C01612 V=800.0 PL=0
MOVL C01613 V=800.0 PL=0
MOVL C01614 V=800.0 PL=0
MOVL C01615 V=800.0 PL=0
MOVL C01616 V=800.0 PL=0
MOVL C01617 V=800.0 PL=0
MOVL C01618 V=800.0 PL=0
MOVL C01619 V=800.0 PL=0
MOVL C01620 V=800.0 PL=0
MOVL C01621 V=800.0 PL=0
MOVL C01622 V=800.0 PL=0
MOVL C01623 V=800.0 PL=0
MOVL C01624 V=800.0 PL=0
MOVL C01625 V=800.0 PL=0
MOVL C01626 V=800.0 PL=0
MOVL C01627 V=800.0 PL=0
MOVL C01628 V=800.0 PL=0
MOVL C01629 V=800.0 PL=0
MOVL C01630 V=800.0 PL=0
MOVL C01631 V=800.0 PL=0
MOVL C01632 V=800.0 PL=0
MOVL C01633 V=800.0 PL=0
MOVL C01634 V=800.0 PL=0
MOVL C01635 V=800.0 PL=0
MOVL C01636 V=800.0 PL=0
MOVL C01637 V=800.0 PL=0
MOVL C01638 V=800.0 PL=0
MOVL C01639 V=800.0 PL=0
MOVL C01640 V=800.0 PL=0
MOVL C01641 V=800.0 PL=0
MOVL C01642 V=800.0 PL=0
MOVL C01643 V=800.0 PL=0
MOVL C01644 V=800.0 PL=0
MOVL C01645 V=800.0 PL=0
MOVL C01646 V=800.0 PL=0
MOVL C01647 V=800.0 PL=0
MOVL C01648 V=800.0 PL=0
MOVL C01649 V=800.0 PL=0
MOVL C01650 V=800.0 PL=0
MOVL C01651 V=800.0 PL=0
MOVL C01652 V=800.0 PL=0
MOVL C01653 V=800.0 PL=0
MOVL C01654 V=800.0 PL=0
MOVL C01655 V=800.0 PL=0
MOVL C01656 V=800.0 PL=0
MOVL C01657 V=800.0 PL=0
MOVL C01658 V=800.0 PL=0
MOVL C01659 V=800.0 PL=0
MOVL C01660 V=800.0 PL=0
MOVL C01661 V=800.0 PL=0
MOVL C01662 V=800.0 PL=0
MOVL C01663 V=800.0 PL=0
MOVL C01664 V=800.0 PL=0
MOVL C01665 V=800.0 PL=0
MOVL C01666 V=800.0 PL=0
MOVL C01667 V=800.0 PL=0
MOVL C01668 V=800.0 PL=0
MOVL C01669 V=800.0 PL=0
MOVL C01670 V=800.0 PL=0
MOVL C01671 V=800.0 PL=0
MOVL C01672 V=800.0 PL=0
MOVL C01673 V=800.0 PL=0
MOVL C01674 V=800.0 PL=0
MOVL C01675 V=800.0 PL=0
MOVL C01676 V=800.0 PL=0
MOVL C01677 V=800.0 PL=0
MOVL C01678 V=800.0 PL=0
MOVL C01679 V=800.0 PL=0
MOVL C01680 V=800.0 PL=0
MOVL C01681 V=800.0 PL=0
MOVL C01682 V=800.0 PL=0
MOVL C01683 V=800.0 PL=0
MOVL C01684 V=800.0 PL=0
MOVL C01685 V=800.0 PL=0
MOVL C01686 V=800.0 PL=0
MOVL C01687 V=800.0 PL=0
MOVL C01688 V=800.0 PL=0
MOVL C01689 V=800.0 PL=0
MOVL C01690 V=800.0 PL=0
MOVL C01691 V=800.0 PL=0
MOVL C01692 V=800.0 PL=0
MOVL C01693 V=800.0 PL=0
MOVL C01694 V=800.0 PL=0
MOVL C01695 V=800.0 PL=0
MOVL C01696 V=800.0 PL=0
MOVL C01697 V=800.0 PL=0
MOVL C01698 V=800.0 PL=0
MOVL C01699 V=800.0 PL=0
MOVL C01700 V=800.0 PL=0
MOVL C01701 V=800.0 PL=0
MOVL C01702 V=800.0 PL=0
MOVL C01703 V=800.0 PL=0
MOVL C01704 V=800.0 PL=0
MOVL C01705 V=800.0 PL=0
MOVL C01706 V=800.0 PL=0
MOVL C01707 V=800.0 PL=0
MOVL C01708 V=800.0 PL=0
MOVL C01709 V=800.0 PL=0
MOVL C01710 V=800.0 PL=0
MOVL C01711 V=800.0 PL=0
MOVL C01712 V=800.0 PL=0
MOVL C01713 V=800.0 PL=0
MOVL C01714 V=800.0 PL=0
MOVL C01715 V=800.0 PL=0
MOVL C01716 V=800.0 PL=0
MOVL C01717 V=800.0 PL=0
MOVL C01718 V=800.0 PL=0
MOVL C01719 V=800.0 PL=0
MOVL C01720 V=800.0 PL=0
MOVL C01721 V=800.0 PL=0
MOVL C01722 V=800.0 PL=0
MOVL C01723 V=800.0 PL=0
MOVL C01724 V=800.0 PL=0
MOVL C01725 V=800.0 PL=0
MOVL C01726 V=800.0 PL=0
MOVL C01727 V=800.0 PL=0
MOVL C01728 V=800.0 PL=0
MOVL C01729 V=800.0 PL=0
MOVL C01730 V=800.0 PL=0
MOVL C01731 V=800.0 PL=0
MOVL C01732 V=800.0 PL=0
MOVL C01733 V=800.0 PL=0
MOVL C01734 V=800.0 PL=0
MOVL C01735 V=800.0 PL=0
MOVL C01736 V=800.0 PL=0
MOVL C01737 V=800.0 PL=0
MOVL C01738 V=800.0 PL=0
MOVL C01739 V=800.0 PL=0
MOVL C01740 V=800.0 PL=0
MOVL C01741 V=800.0 PL=0
MOVL C01742 V=800.0 PL=0
MOVL C01743 V=800.0 PL=0
MOVL C01744 V=800.0 PL=0
MOVL C01745 V=800.0 PL=0
MOVL C01746 V=800.0 PL=0
MOVL C01747 V=800.0 PL=0
MOVL C01748 V=800.0 PL=0
MOVL C01749 V=800.0 PL=0
MOVL C01750 V=800.0 PL=0
MOVL C01751 V=800.0 PL=0
MOVL C01752 V=800.0 PL=0
MOVL C01753 V=800.0 PL=0
MOVL C01754 V=800.0 PL=0
MOVL C01755 V=800.0 PL=0
MOVL C01756 V=800.0 PL=0
MOVL C01757 V=800.0 PL=0
MOVL C01758 V=800.0 PL=0
MOVL C01759 V=800.0 PL=0
MOVL C01760 V=800.0 PL=0
MOVL C01761 V=800.0 PL=0
MOVL C01762 V=800.0 PL=0
MOVL C01763 V=800.0 PL=0
MOVL C01764 V=800.0 PL=0
MOVL C01765 V=800.0 PL=0
MOVL C01766 V=800.0 PL=0
MOVL C01767 V=800.0 PL=0
MOVL C01768 V=800.0 PL=0
MOVL C01769 V=800.0 PL=0
MOVL C01770 V=800.0 PL=0
MOVL C01771 V=800.0 PL=0
MOVL C01772 V=800.0 PL=0
MOVL C01773 V=800.0 PL=0
MOVL C01774 V=800.0 PL=0
MOVL C01775 V=800.0 PL=0
MOVL C01776 V=800.0 PL=0
MOVL C01777 V=800.0 PL=0
MOVL C01778 V=800.0 PL=0
MOVL C01779 V=800.0 PL=0
MOVL C01780 V=800.0 PL=0
MOVL C01781 V=800.0 PL=0
MOVL C01782 V=800.0 PL=0
MOVL C01783 V=800.0 PL=0
MOVL C01784 V=800.0 PL=0
MOVL C01785 V=800.0 PL=0
MOVL C01786 V=800.0 PL=0
MOVL C01787 V=800.0 PL=0
MOVL C01788 V=800.0 PL=0
MOVL C01789 V=800.0 PL=0
MOVL C01790 V=800.0 PL=0
MOVL C01791 V=800.0 PL=0
MOVL C01792 V=800.0 PL=0
MOVL C01793 V=800.0 PL=0
MOVL C01794 V=800.0 PL=0
MOVL C01795 V=800.0 PL=0
MOVL C01796 V=800.0 PL=0
MOVL C01797 V=800.0 PL=0
MOVL C01798 V=800.0 PL=0
MOVL C01799 V=800.0 PL=0
MOVL C01800 V=800.0 PL=0
MOVL C01801 V=800.0 PL=0
MOVL C01802 V=800.0 PL=0
MOVL C01803 V=800.0 PL=0
MOVL C01804 V=800.0 PL=0
MOVL C01805 V=800.0 PL=0
MOVL C01806 V=800.0 PL=0
MOVL C01807 V=800.0 PL=0
MOVL C01808 V=800.0 PL=0
MOVL C01809 V=800.0 PL=0
MOVL C01810 V=800.0 PL=0
MOVL C01811 V=800.0 PL=0
MOVL C01812 V=800.0 PL=0
MOVL C01813 V=800.0 PL=0
MOVL C01814 V=800.0 PL=0
MOVL C01815 V=800.0 PL=0
MOVL C01816 V=800.0 PL=0
MOVL C01817 V=800.0 PL=0
MOVL C01818 V=800.0 PL=0
MOVL C01819 V=800.0 PL=0
MOVL C01820 V=800.0 PL=0
MOVL C01821 V=800.0 PL=0
MOVL C01822 V=800.0 PL=0
MOVL C01823 V=800.0 PL=0
MOVL C01824 V=800.0 PL=0
MOVL C01825 V=800.0 PL=0
MOVL C01826 V=800.0 PL=0
MOVL C01827 V=800.0 PL=0
MOVL C01828 V=800.0 PL=0
MOVL C01829 V=800.0 PL=0
MOVL C01830 V=800.0 PL=0
MOVL C01831 V=800.0 PL=0
MOVL C01832 V=800.0 PL=0
MOVL C01833 V=800.0 PL=0
MOVL C01834 V=800.0 PL=0
MOVL C01835 V=800.0 PL=0
MOVL C01836 V=800.0 PL=0
MOVL C01837 V=800.0 PL=0
MOVL C01838 V=800.0 PL=0
MOVL C01839 V=800.0 PL=0
MOVL C01840 V=800.0 PL=0
MOVL C01841 V=800.0 PL=0
MOVL C01842 V=800.0 PL=0
MOVL C01843 V=800.0 PL=0
MOVL C01844 V=800.0 PL=0
MOVL C01845 V=800.0 PL=0
MOVL C01846 V=800.0 PL=0
MOVL C01847 V=800.0 PL=0
MOVL C01848 V=800.0 PL=0
MOVL C01849 V=800.0 PL=0
MOVL C01850 V=800.0 PL=0
MOVL C01851 V=800.0 PL=0
MOVL C01852 V=800.0 PL=0
MOVL C01853 V=800.0 PL=0
MOVL C01854 V=800.0 PL=0
MOVL C01855 V=800.0 PL=0
MOVL C01856 V=800.0 PL=0
MOVL C01857 V=800.0 PL=0
MOVL C01858 V=800.0 PL=0
MOVL C01859 V=800.0 PL=0
MOVL C01860 V=800.0 PL=0
MOVL C01861 V=800.0 PL=0
MOVL C01862 V=800.0 PL=0
MOVL C01863 V=800.0 PL=0
MOVL C01864 V=800.0 PL=0
MOVL C01865 V=800.0 PL=0
MOVL C01866 V=800.0 PL=0
MOVL C01867 V=800.0 PL=0
MOVL C01868 V=800.0 PL=0
MOVL C01869 V=800.0 PL=0
MOVL C01870 V=800.0 PL=0
MOVL C01871 V=800.0 PL=0
MOVL C01872 V=800.0 PL=0
MOVL C01873 V=800.0 PL=0
MOVL C01874 V=800.0 PL=0
MOVL C01875 V=800.0 PL=0
MOVL C01876 V=800.0 PL=0
MOVL C01877 V=800.0 PL=0
MOVL C01878 V=800.0 PL=0
MOVL C01879 V=800.0 PL=0
MOVL C01880 V=800.0 PL=0
MOVL C01881 V=800.0 PL=0
MOVL C01882 V=800.0 PL=0
MOVL C01883 V=800.0 PL=0
MOVL C01884 V=800.0 PL=0
MOVL C01885 V=800.0 PL=0
MOVL C01886 V=800.0 PL=0
MOVL C01887 V=800.0 PL=0
MOVL C01888 V=800.0 PL=0
MOVL C01889 V=800.0 PL=0
MOVL C01890 V=800.0 PL=0
MOVL C01891 V=800.0 PL=0
MOVL C01892 V=800.0 PL=0
MOVL C01893 V=800.0 PL=0
MOVL C01894 V=800.0 PL=0
MOVL C01895 V=800.0 PL=0
MOVL C01896 V=800.0 PL=0
MOVL C01897 V=800.0 PL=0
MOVL C01898 V=800.0 PL=0
MOVL C01899 V=800.0 PL=0
MOVL C01900 V=800.0 PL=0
MOVL C01901 V=800.0 PL=0
MOVL C01902 V=800.0 PL=0
MOVL C01903 V=800.0 PL=0
MOVL C01904 V=800.0 PL=0
MOVL C01905 V=800.0 PL=0
MOVL C01906 V=800.0 PL=0
MOVL C01907 V=800.0 PL=0
MOVL C01908 V=800.0 PL=0
MOVL C01909 V=800.0 PL=0
MOVL C01910 V=800.0 PL=0
MOVL C01911 V=800.0 PL=0
MOVL C01912 V=800.0 PL=0
MOVL C01913 V=800.0 PL=0
MOVL C01914 V=800.0 PL=0
MOVL C01915 V=800.0 PL=0
MOVL C01916 V=800.0 PL=0
MOVL C01917 V=800.0 PL=0
MOVL C01918 V=800.0 PL=0
MOVL C01919 V=800.0 PL=0
MOVL C01920 V=800.0 PL=0
MOVL C01921 V=800.0 PL=0
MOVL C01922 V=800.0 PL=0
MOVL C01923 V=800.0 PL=0
MOVL C01924 V=800.0 PL=0
MOVL C01925 V=800.0 PL=0
MOVL C01926 V=800.0 PL=0
MOVL C01927 V=800.0 PL=0
MOVL C01928 V=800.0 PL=0
MOVL C01929 V=800.0 PL=0
MOVL C01930 V=800.0 PL=0
MOVL C01931 V=800.0 PL=0
MOVL C01932 V=800.0 PL=0
MOVL C01933 V=800.0 PL=0
MOVL C01934 V=800.0 PL=0
MOVL C01935 V=800.0 PL=0
MOVL C01936 V=800.0 PL=0
MOVL C01937 V=800.0 PL=0
MOVL C01938 V=800.0 PL=0
MOVL C01939 V=800.0 PL=0
MOVL C01940 V=800.0 PL=0
MOVL C01941 V=800.0 PL=0
MOVL C01942 V=800.0 PL=0
MOVL C01943 V=800.0 PL=0
MOVL C01944 V=800.0 PL=0
MOVL C01945 V=800.0 PL=0
MOVL C01946 V=800.0 PL=0
MOVL C01947 V=800.0 PL=0
MOVL C01948 V=800.0 PL=0
MOVL C01949 V=800.0 PL=0
MOVL C01950 V=800.0 PL=0
MOVL C01951 V=800.0 PL=0
MOVL C01952 V=800.0 PL=0
MOVL C01953 V=800.0 PL=0
MOVL C01954 V=800.0 PL=0
MOVL C01955 V=800.0 PL=0
MOVL C01956 V=800.0 PL=0
MOVL C01957 V=800.0 PL=0
MOVL C01958 V=800.0 PL=0
MOVL C01959 V=800.0 PL=0
MOVL C01960 V=800.0 PL=0
MOVL C01961 V=800.0 PL=0
MOVL C01962 V=800.0 PL=0
MOVL C01963 V=800.0 PL=0
MOVL C01964 V=800.0 PL=0
MOVL C01965 V=800.0 PL=0
MOVL C01966 V=800.0 PL=0
MOVL C01967 V=800.0 PL=0
MOVL C01968 V=800.0 PL=0
MOVL C01969 V=800.0 PL=0
MOVL C01970 V=800.0 PL=0
MOVL C01971 V=800.0 PL=0
MOVL C01972 V=800.0 PL=0
MOVL C01973 V=800.0 PL=0
MOVL C01974 V=800.0 PL=0
MOVL C01975 V=800.0 PL=0
MOVL C01976 V=800.0 PL=0
MOVL C01977 V=800.0 PL=0
MOVL C01978 V=800.0 PL=0
MOVL C01979 V=800.0 PL=0
MOVL C01980 V=800.0 PL=0
MOVL C01981 V=800.0 PL=0
MOVL C01982 V=800.0 PL=0
MOVL C01983 V=800.0 PL=0
MOVL C01984 V=800.0 PL=0
MOVL C01985 V=800.0 PL=0
MOVL C01986 V=800.0 PL=0
MOVL C01987 V=800.0 PL=0
MOVL C01988 V=800.0 PL=0
MOVL C01989 V=800.0 PL=0
MOVL C01990 V=800.0 PL=0
MOVL C01991 V=800.0 PL=0
MOVL C01992 V=800.0 PL=0
MOVL C01993 V=800.0 PL=0
MOVL C01994 V=800.0 PL=0
MOVL C01995 V=800.0 PL=0
MOVL C01996 V=800.0 PL=0
MOVL C01997 V=800.0 PL=0
MOVL C01998 V=800.0 PL=0
MOVL C01999 V=800.0 PL=0
MOVL C02000 V=800.0 PL=0
MOVL C02001 V=800.0 PL=0
MOVL C02002 V=800.0 PL=0
MOVL C02003 V=800.0 PL=0
MOVL C02004 V=800.0 PL=0
MOVL C02005 V=800.0 PL=0
MOVL C02006 V=800.0 PL=0
MOVL C02007 V=800.0 PL=0
MOVL C02008 V=800.0 PL=0
MOVL C02009 V=800.0 PL=0
MOVL C02010 V=800.0 PL=0
MOVL C02011 V=800.0 PL=0
MOVL C02012 V=800.0 PL=0
MOVL C02013 V=800.0 PL=0
MOVL C02014 V=800.0 PL=0
MOVL C02015 V=800.0 PL=0
MOVL C02016 V=800.0 PL=0
MOVL C02017 V=800.0 PL=0
MOVL C02018 V=800.0 PL=0
MOVL C02019 V=800.0 PL=0
MOVL C02020 V=800.0 PL=0
MOVL C02021 V=800.0 PL=0
MOVL C02022 V=800.0 PL=0
MOVL C02023 V=800.0 PL=0
MOVL C02024 V=800.0 PL=0
MOVL C02025 V=800.0 PL=0
MOVL C02026 V=800.0 PL=0
MOVL C02027 V=800.0 PL=0
MOVL C02028 V=800.0 PL=0
MOVL C02029 V=800.0 PL=0
MOVL C02030 V=800.0 PL=0
MOVL C02031 V=800.0 PL=0
MOVL C02032 V=800.0 PL=0
MOVL C02033 V=800.0 PL=0
MOVL C02034 V=800.0 PL=0
MOVL C02035 V=800.0 PL=0
MOVL C02036 V=800.0 PL=0
MOVL C02037 V=800.0 PL=0
MOVL C02038 V=800.0 PL=0
MOVL C02039 V=800.0 PL=0
MOVL C02040 V=800.0 PL=0
MOVL C02041 V=800.0 PL=0
MOVL C02042 V=800.0 PL=0
MOVL C02043 V=800.0 PL=0
MOVL C02044 V=800.0 PL=0
MOVL C02045 V=800.0 PL=0
MOVL C02046 V=800.0 PL=0
MOVL C02047 V=800.0 PL=0
MOVL C02048 V=800.0 PL=0
MOVL C02049 V=800.0 PL=0
MOVL C02050 V=800.0 PL=0
MOVL C02051 V=800.0 PL=0
MOVL C02052 V=800.0 PL=0
MOVL C02053 V=800.0 PL=0
MOVL C02054 V=800.0 PL=0
MOVL C02055 V=800.0 PL=0
MOVL C02056 V=800.0 PL=0
MOVL C02057 V=800.0 PL=0
MOVL C02058 V=800.0 PL=0
MOVL C02059 V=800.0 PL=0
MOVL C02060 V=800.0 PL=0
MOVL C02061 V=800.0 PL=0
MOVL C02062 V=800.0 PL=0
MOVL C02063 V=800.0 PL=0
MOVL C02064 V=800.0 PL=0
MOVL C02065 V=800.0 PL=0
MOVL C02066 V=800.0 PL=0
MOVL C02067 V=800.0 PL=0
MOVL C02068 V=800.0 PL=0
MOVL C02069 V=800.0 PL=0
MOVL C02070 V=800.0 PL=0
MOVL C02071 V=800.0 PL=0
MOVL C02072 V=800.0 PL=0
MOVL C02073 V=800.0 PL=0
MOVL C02074 V=800.0 PL=0
MOVL C02075 V=800.0 PL=0
MOVL C02076 V=800.0 PL=0
MOVL C02077 V=800.0 PL=0
MOVL C02078 V=800.0 PL=0
MOVL C02079 V=800.0 PL=0
MOVL C02080 V=800.0 PL=0
MOVL C02081 V=800.0 PL=0
MOVL C02082 V=800.0 PL=0
MOVL C02083 V=800.0 PL=0
MOVL C02084 V=800.0 PL=0
MOVL C02085 V=800.0 PL=0
MOVL C02086 V=800.0 PL=0
MOVL C02087 V=800.0 PL=0
MOVL C02088 V=800.0 PL=0
MOVL C02089 V=800.0 PL=0
MOVL C02090 V=800.0 PL=0
MOVL C02091 V=800.0 PL=0
MOVL C02092 V=800.0 PL=0
MOVL C02093 V=800.0 PL=0
MOVL C02094 V=800.0 PL=0
